# B&R Automation Studio project NAEUL004C00R13L518F00 (part 42)

#### Act_InitGlobal.st
```iecst
(** 2019-04-09 **)
ACTION Act_InitGlobal:

	(* Always Change If Project Change *)

	//Pass Data To Link
	p_bLinkOpsRun ACCESS p_OpsRun;

	p_bLinkDISafetyRlySig ACCESS p_DISafetyRlySig;
	p_bLinkDIConvClrSen ACCESS p_DIConvClrSen;
	p_bLinkDIPusherRetRS ACCESS p_DIPusherRetRS;
	p_bConvPusherReachedRetSlw ACCESS p_PshrConvPshrRetAllwTrav;
	p_eLinkLifterBtmStat ACCESS p_LifterBtmStat;
	p_eLinkLifterBtmStatus ACCESS p_LifterBtmStatus;
	p_eLinkLifter2Stat ACCESS p_Lifter2Stat;
	p_eLinkLifter2Status ACCESS p_Lifter2Status;

	//Pass Data To Internal Use
	p_udiRstErr ACCESS p_RstErrReset;
	p_bPrep ACCESS p_NtParamProjOutletShut2Prep;
	p_bUISimu ACCESS p_UISimuMod;
	p_bManual ACCESS p_UIMnlMod;
	p_bSimu ACCESS p_SimuRun;
	p_bTwoCtrlIn ACCESS p_NtParamOutShutterTwoCtrlIn;
	p_sProgNm ACCESS p_NtParamOutShutterProgNm;
	p_bExtSen ACCESS p_DIOutShutterCloseRS2;
	p_bRetSen ACCESS p_DIOutShutterOpenRS2;
	p_tExtTO ACCESS p_NtParamOutShutterExtTO;
	p_tRetTO ACCESS p_NtParamOutShutterRetTO;
	p_bNtSettingsLoadDone ACCESS p_StartupNtSettingsLoadDone;
	p_bNtParamProjLifter2Prep ACCESS p_NtParamProjLifter2Prep;
	(* Always Change If Project Change *)

END_ACTION
```

#### Act_LinkAction.st
```iecst
(** 2019-04-09 **)
ACTION Act_LinkAction:

	IF p_bLinkOpsRun = TRUE THEN
		IF p_bNtParamProjLifter2Prep = FALSE  THEN
			IF p_eLinkLifterBtmStat = LifterActIdle AND p_eLinkLifterBtmStatus <> Busy  THEN //
				p_eAct ACCESS p_OpsTravLifULOutletPneuAct2;
			ELSE
				p_eAct ACCESS ADR(eAct);
			END_IF
		ELSE
			IF p_eLinkLifterBtmStat = LifterActIdle AND p_eLinkLifterBtmStatus <> Busy AND p_eLinkLifter2Stat = LifterActIdle AND p_eLinkLifter2Status <> Busy  THEN // p_eLinkLifter2Status <> Busy
				p_eAct ACCESS p_OpsTravLifULOutletPneuAct2;
			ELSE
				p_eAct ACCESS ADR(eAct);
			END_IF
		END_IF
	ELSIF p_bManual = TRUE OR p_bUISimu THEN
		p_eAct ACCESS p_UIOutShutterAct2;
	ELSIF p_bSimu THEN
		p_eAct ACCESS p_Simu1OutShutterAct2;
	ELSE
		p_eAct ACCESS ADR(eAct);
	END_IF

END_ACTION
```

#### Act_LinkEn.st
```iecst
(** 2019-01-11 **)
ACTION Act_LinkEn:

	//Link bPrep, bEn & bDis
	p_bEn ACCESS p_NtParamCurtainSenPrep;

END_ACTION
```

#### Init.st
```iecst
(** 2019-03-25 **)
PROGRAM _INIT

	(* Always Change If Project Change *)

	//Pass Address To Global Address For External Use
	//Action, State & Status
	p_Pneu2SenOutShutterStat2		:= ADR(eStat);
	p_Pneu2SenOutShutterStatus2		:= ADR(eStatus);
	p_Pneu2SenOutShutterStatTxt2	:= ADR(sStatTxt);

	//Alarm
	p_Pneu2SenOutShutterAlmData2	:= ADR(tyAlmData);

	//Output
	p_Pneu2SenOutShutterExtCtrl2	:= ADR(bExtCtrl);
	p_Pneu2SenOutShutterRetCtrl2	:= ADR(bRetCtrl);
	p_Pneu2SenOutShutterTwoCtrlOut2	:= ADR(bTwoCtrlOut);
	p_Pneu2SenOutShutterExtended2	:= ADR(bExtended);
	p_Pneu2SenOutShutterRetracted2	:= ADR(bRetracted);

	(* Always Change If Project Change *)

END_PROGRAM
```

### Program Logical/Pneu/Pneu2SenOutShutter3

#### InputRef_Link.var
```iecst
(*2019-04-09*)
(**)
(*External*)
VAR
	p_bLinkOpsRun : REFERENCE TO BOOL;
END_VAR
(**)
VAR
	p_bLinkDISafetyRlySig : REFERENCE TO BOOL;
	p_bLinkDIConvClrSen : REFERENCE TO BOOL;
	p_bLinkDIPusherRetRS : REFERENCE TO BOOL;
	p_bConvPusherReachedRetSlw : REFERENCE TO BOOL;
	p_eLinkLifter2Stat : REFERENCE TO eLifterAction;
	p_eLinkLifter2Status : REFERENCE TO eFBStatus;
	p_eLinkLifterBtmStat : REFERENCE TO eLifterAction;
	p_eLinkLifterBtmStatus : REFERENCE TO eFBStatus;
END_VAR
```

#### Act_Alarm.st
```iecst
(** 2019-03-25 **)
ACTION Act_Alarm:

	//Error
	IF EDGEPOS(eStatus = Error) THEN

		tyAlmData.sProgNm		:= p_sProgNm;
		tyAlmData.udiCode		:= udiStatus;
		tyAlmData.eSeverity		:= AlmSeverityError;
		tyAlmData.udiRunTime	:= tyAlmData.udiRunTime + 1;
		tyAlmData.bAlm			:= TRUE;
		tyAlmData.udiModuleNum  := udiModuleNum;
		g_sPneu2SenProgNm		:= p_sProgNm;

		//Get Error Message
		IF tyAlmData.udiCode < 10000 OR tyAlmData.udiCode > 10099 THEN
			tyAlmData.sAlmMsg	:= 'Unknown';
			tyAlmData.sRcyMsg	:= 'Unknown';
		ELSE
			tyAlmData.sAlmMsg	:= a_tyAlmText[tyAlmData.udiCode].sAlmText;
			tyAlmData.sRcyMsg	:= a_tyAlmText[tyAlmData.udiCode].sRcyText;
		END_IF

		sStatTxt	:= tyAlmData.sAlmMsg;

	ELSIF bRstErr AND (tyAlmData.udiCode <> 0) THEN

		tyAlmData.udiCode	:= 0;
		tyAlmData.eSeverity	:= AlmSeverityNA;
		tyAlmData.sAlmMsg	:= '';
		tyAlmData.sRcyMsg	:= '';
		tyAlmData.bAlm			:= FALSE;
		sStatTxt	:= a_sStatText[eStat];

	END_IF

END_ACTION
```

#### Act_InitGlobal.st
```iecst
(** 2019-04-09 **)
ACTION Act_InitGlobal:

	(* Always Change If Project Change *)

	//Pass Data To Link
	p_bLinkOpsRun ACCESS p_OpsRun;

	p_bLinkDISafetyRlySig ACCESS p_DISafetyRlySig;
	p_bLinkDIConvClrSen ACCESS p_DIConvClrSen;
	p_bLinkDIPusherRetRS ACCESS p_DIPusherRetRS;
	p_bConvPusherReachedRetSlw ACCESS p_PshrConvPshrRetAllwTrav;
	p_eLinkLifterBtmStat ACCESS p_LifterBtmStat;
	p_eLinkLifterBtmStatus ACCESS p_LifterBtmStatus;
	p_eLinkLifter2Stat ACCESS p_Lifter2Stat;
	p_eLinkLifter2Status ACCESS p_Lifter2Status;

	//Pass Data To Internal Use
	p_udiRstErr ACCESS p_RstErrReset;
	p_bPrep ACCESS p_NtParamProjOutletShut3Prep;
	p_bUISimu ACCESS p_UISimuMod;
	p_bManual ACCESS p_UIMnlMod;
	p_bSimu ACCESS p_SimuRun;
	p_bTwoCtrlIn ACCESS p_NtParamOutShutterTwoCtrlIn;
	p_sProgNm ACCESS p_NtParamOutShutterProgNm;
	p_bExtSen ACCESS p_DIOutShutterCloseRS3;
	p_bRetSen ACCESS p_DIOutShutterOpenRS3;
	p_tExtTO ACCESS p_NtParamOutShutterExtTO;
	p_tRetTO ACCESS p_NtParamOutShutterRetTO;
	p_bNtSettingsLoadDone ACCESS p_StartupNtSettingsLoadDone;
	p_bNtParamProjLifter2Prep ACCESS p_NtParamProjLifter2Prep;
	(* Always Change If Project Change *)

END_ACTION
```

#### Act_Link.st
```iecst
(** 2019-03-29 **)
ACTION Act_Link:

	p_bExtSafetySen := (p_bLinkDIConvClrSen = FALSE) AND (p_bLinkDIPusherRetRS OR p_bConvPusherReachedRetSlw);

	IF p_bLinkDISafetyRlySig = FALSE THEN
		bExtCtrl	:= FALSE;
		bRetCtrl	:= FALSE;
		bExtended	:= FALSE;
		bRetracted	:= FALSE;
	END_IF

END_ACTION
```

#### Act_LinkAction.st
```iecst
(** 2019-04-09 **)
ACTION Act_LinkAction:

	IF p_bLinkOpsRun = TRUE THEN
		IF p_bNtParamProjLifter2Prep = FALSE  THEN
			IF p_eLinkLifterBtmStat = LifterActIdle AND p_eLinkLifterBtmStatus <> Busy  THEN //
				p_eAct ACCESS p_OpsTravLifULOutletPneuAct3;
			ELSE
				p_eAct ACCESS ADR(eAct);
			END_IF
		ELSE
			IF p_eLinkLifterBtmStat = LifterActIdle AND p_eLinkLifterBtmStatus <> Busy AND p_eLinkLifter2Stat = LifterActIdle AND p_eLinkLifter2Status <> Busy  THEN // p_eLinkLifter2Status <> Busy
				p_eAct ACCESS p_OpsTravLifULOutletPneuAct3;
			ELSE
				p_eAct ACCESS ADR(eAct);
			END_IF
		END_IF
	ELSIF p_bManual = TRUE OR p_bUISimu THEN
		p_eAct ACCESS p_UIOutShutterAct3;
	ELSIF p_bSimu THEN
		p_eAct ACCESS p_Simu1OutShutterAct3;
	ELSE
		p_eAct ACCESS ADR(eAct);
	END_IF

END_ACTION
```

### Program Logical/Pneu/Pneu2SenSelClamp1

#### Act_InitGlobal.st
```iecst
(** 2019-04-09 **)
ACTION Act_InitGlobal:

	(* Always Change If Project Change *)

	//Pass Data To Link
	p_bLinkOpsRun ACCESS p_OpsRun;

	p_bLinkDISafetyRlySig ACCESS p_DISafetyRlySig;

	//Pass Data To Internal Use
	p_udiRstErr ACCESS p_RstErrReset;
	p_bPrep ACCESS p_NtParamProjMagAutoVerifyPrep;
	p_bManual ACCESS p_UIMnlMod;
	p_bTwoCtrlIn ACCESS p_NtParamSelClamp1TwoCtrlIn;
	p_sProgNm ACCESS p_NtParamSelClamp1ProgNm;
	p_bExtSen ACCESS p_DIMag1SelUnclampRS;
//	p_bRetSen ACCESS p_DIOutShutterOpenRS;
	p_tExtTO ACCESS p_NtParamSelClamp1ExtDlyTm;
	p_tRetTO ACCESS p_NtParamSelClamp1RetDlyTm;
	p_bNtSettingsLoadDone ACCESS p_StartupNtSettingsLoadDone;

	(* Always Change If Project Change *)

END_ACTION
```

#### Act_LinkAction.st
```iecst
(** 2019-04-09 **)
ACTION Act_LinkAction:

	IF p_bLinkOpsRun = TRUE THEN
		p_eAct ACCESS p_OpsMagConvUL1StepSelClampCtrl;
	ELSIF p_bManual = TRUE THEN
		p_eAct ACCESS p_UIMagConvSelClp1Act;
	ELSE
		p_eAct ACCESS ADR(eAct);
	END_IF

END_ACTION
```

#### Init.st
```iecst
(** 2019-03-25 **)
PROGRAM _INIT

	(* Always Change If Project Change *)

	//Pass Address To Global Address For External Use
	//Action, State & Status
	p_PneuNoSenSelClamp1Stat		:= ADR(eStat);
	p_PneuNoSenSelClamp1Status		:= ADR(eStatus);
	p_PneuNoSenSelClamp1StatTxt		:= ADR(sStatTxt);

	//Alarm
	p_PneuNoSenSelClamp1AlmData		:= ADR(tyAlmData);

	//Output
	p_PneuNoSenSelClamp1ExtCtrl		:= ADR(bExtCtrl);
	p_PneuNoSenSelClamp1RetCtrl		:= ADR(bRetCtrl);
	p_PneuNoSenSelClamp1TwoCtrlOut	:= ADR(bTwoCtrlOut);
	p_PneuNoSenSelClamp1Extended	:= ADR(bExtended);
	p_PneuNoSenSelClamp1Retracted	:= ADR(bRetracted);

	(* Always Change If Project Change *)

END_PROGRAM
```

### Program Logical/Pneu/Pneu2SenSelClamp2

#### Act_Alarm.st
```iecst
(** 2019-03-25 **)
ACTION Act_Alarm:

	//Error
	IF EDGEPOS(eStatus = Error) THEN

		tyAlmData.sProgNm		:= p_sProgNm;
		tyAlmData.udiCode		:= udiStatus;
		tyAlmData.eSeverity		:= AlmSeverityError;
		tyAlmData.udiRunTime	:= tyAlmData.udiRunTime + 1;
		tyAlmData.bAlm			:= TRUE;
		tyAlmData.udiModuleNum  := udiModuleNum;
		g_sPneu2SenProgNm		:= p_sProgNm;

		//Get Error Message
		IF tyAlmData.udiCode < 10000 OR tyAlmData.udiCode > 10099 THEN
			tyAlmData.sAlmMsg	:= 'Unknown';
			tyAlmData.sRcyMsg	:= 'Unknown';
		ELSE
			tyAlmData.sAlmMsg	:= a_tyAlmText[tyAlmData.udiCode].sAlmText;
			tyAlmData.sRcyMsg	:= a_tyAlmText[tyAlmData.udiCode].sRcyText;
		END_IF

		sStatTxt	:= tyAlmData.sAlmMsg;

	ELSIF bRstErr AND (tyAlmData.udiCode <> 0) THEN

		tyAlmData.udiCode	:= 0;
		tyAlmData.eSeverity	:= AlmSeverityNA;
		tyAlmData.sAlmMsg	:= '';
		tyAlmData.sRcyMsg	:= '';
		tyAlmData.bAlm			:= FALSE;
		sStatTxt	:= a_sStatText[eStat];

	END_IF

END_ACTION
```

#### Act_InitGlobal.st
```iecst
(** 2029-04-09 **)
ACTION Act_InitGlobal:

	(* Always Change If Project Change *)

	//Pass Data To Link
	p_bLinkOpsRun ACCESS p_OpsRun;

	p_bLinkDISafetyRlySig ACCESS p_DISafetyRlySig;

	//Pass Data To Internal Use
	p_udiRstErr ACCESS p_RstErrReset;
	p_bPrep ACCESS p_NtParamProjMagAutoVerifyPrep;
	p_bManual ACCESS p_UIMnlMod;
	p_bTwoCtrlIn ACCESS p_NtParamSelClamp2TwoCtrlIn;
	p_sProgNm ACCESS p_NtParamSelClamp2ProgNm;
	p_bExtSen ACCESS p_DIMag2SelUnclampRS;
//	p_bRetSen ACCESS p_DIOutShutterOpenRS;
	p_tExtTO ACCESS p_NtParamSelClamp2ExtDlyTm;
	p_tRetTO ACCESS p_NtParamSelClamp2RetDlyTm;
	p_bNtSettingsLoadDone ACCESS p_StartupNtSettingsLoadDone;

	(* Always Change If Project Change *)

END_ACTION
```

#### Act_Link.st
```iecst
(** 2019-03-29 **)
ACTION Act_Link:

	IF p_bLinkDISafetyRlySig = FALSE THEN
		bExtCtrl	:= FALSE;
		bRetCtrl	:= FALSE;
		bExtended	:= FALSE;
		bRetracted	:= FALSE;
	END_IF

	p_bRetSen := NOT(p_bExtSen);
END_ACTION
```

#### Act_LinkAction.st
```iecst
(** 2019-04-09 **)
ACTION Act_LinkAction:

	IF p_bLinkOpsRun = TRUE THEN
		p_eAct ACCESS p_OpsMagConvUL2StepSelClampCtrl;
	ELSIF p_bManual = TRUE THEN
		p_eAct ACCESS p_UIMagConvSelClp2Act;
	ELSE
		p_eAct ACCESS ADR(eAct);
	END_IF

END_ACTION
```

#### Init.st
```iecst
(** 2029-03-25 **)
PROGRAM _INIT

	(* Always Change If Project Change *)

	//Pass Address To Global Address For External Use
	//Action, State & Status
	p_PneuNoSenSelClamp2Stat		:= ADR(eStat);
	p_PneuNoSenSelClamp2Status		:= ADR(eStatus);
	p_PneuNoSenSelClamp2StatTxt		:= ADR(sStatTxt);

	//Alarm
	p_PneuNoSenSelClamp2AlmData		:= ADR(tyAlmData);

	//Output
	p_PneuNoSenSelClamp2ExtCtrl		:= ADR(bExtCtrl);
	p_PneuNoSenSelClamp2RetCtrl		:= ADR(bRetCtrl);
	p_PneuNoSenSelClamp2TwoCtrlOut	:= ADR(bTwoCtrlOut);
	p_PneuNoSenSelClamp2Extended	:= ADR(bExtended);
	p_PneuNoSenSelClamp2Retracted	:= ADR(bRetracted);

	(* Always Change If Project Change *)

END_PROGRAM
```

### Program Logical/Pneu/Pneu2SenSelClamp3

#### Act_Alarm.st
```iecst
(** 2019-03-25 **)
ACTION Act_Alarm:

	//Error
	IF EDGEPOS(eStatus = Error) THEN

		tyAlmData.sProgNm		:= p_sProgNm;
		tyAlmData.udiCode		:= udiStatus;
		tyAlmData.eSeverity		:= AlmSeverityError;
		tyAlmData.udiRunTime	:= tyAlmData.udiRunTime + 1;
		tyAlmData.bAlm			:= TRUE;
		tyAlmData.udiModuleNum  := udiModuleNum;
		g_sPneu2SenProgNm		:= p_sProgNm;

		//Get Error Message
		IF tyAlmData.udiCode < 10000 OR tyAlmData.udiCode > 10099 THEN
			tyAlmData.sAlmMsg	:= 'Unknown';
			tyAlmData.sRcyMsg	:= 'Unknown';
		ELSE
			tyAlmData.sAlmMsg	:= a_tyAlmText[tyAlmData.udiCode].sAlmText;
			tyAlmData.sRcyMsg	:= a_tyAlmText[tyAlmData.udiCode].sRcyText;
		END_IF

		sStatTxt	:= tyAlmData.sAlmMsg;

	ELSIF bRstErr AND (tyAlmData.udiCode <> 0) THEN

		tyAlmData.udiCode	:= 0;
		tyAlmData.eSeverity	:= AlmSeverityNA;
		tyAlmData.sAlmMsg	:= '';
		tyAlmData.sRcyMsg	:= '';
		tyAlmData.bAlm			:= FALSE;
		sStatTxt	:= a_sStatText[eStat];

	END_IF

END_ACTION
```

#### Act_InitGlobal.st
```iecst
(** 2039-04-09 **)
ACTION Act_InitGlobal:

	(* Always Change If Project Change *)

	//Pass Data To Link
	p_bLinkOpsRun ACCESS p_OpsRun;

	p_bLinkDISafetyRlySig ACCESS p_DISafetyRlySig;

	//Pass Data To Internal Use
	p_udiRstErr ACCESS p_RstErrReset;
	p_bPrep ACCESS p_NtParamProjMagAutoVerifyPrep;
	p_bManual ACCESS p_UIMnlMod;
	p_bTwoCtrlIn ACCESS p_NtParamSelClamp3TwoCtrlIn;
	p_sProgNm ACCESS p_NtParamSelClamp3ProgNm;
	p_bExtSen ACCESS p_DIMag3SelUnclampRS;
//	p_bRetSen ACCESS p_DIOutShutterOpenRS;
	p_tExtTO ACCESS p_NtParamSelClamp3ExtDlyTm;
	p_tRetTO ACCESS p_NtParamSelClamp3RetDlyTm;
	p_bNtSettingsLoadDone ACCESS p_StartupNtSettingsLoadDone;

	(* Always Change If Project Change *)

END_ACTION
```

#### Act_LinkAction.st
```iecst
(** 2019-04-09 **)
ACTION Act_LinkAction:

	IF p_bLinkOpsRun = TRUE THEN
		p_eAct ACCESS p_OpsMagConvUL3StepSelClampCtrl;
	ELSIF p_bManual = TRUE THEN
		p_eAct ACCESS p_UIMagConvSelClp3Act;
	ELSE
		p_eAct ACCESS ADR(eAct);
	END_IF

END_ACTION
```

#### Init.st
```iecst
(** 2039-03-25 **)
PROGRAM _INIT

	(* Always Change If Project Change *)

	//Pass Address To Global Address For External Use
	//Action, State & Status
	p_PneuNoSenSelClamp3Stat		:= ADR(eStat);
	p_PneuNoSenSelClamp3Status		:= ADR(eStatus);
	p_PneuNoSenSelClamp3StatTxt		:= ADR(sStatTxt);

	//Alarm
	p_PneuNoSenSelClamp3AlmData		:= ADR(tyAlmData);

	//Output
	p_PneuNoSenSelClamp3ExtCtrl		:= ADR(bExtCtrl);
	p_PneuNoSenSelClamp3RetCtrl		:= ADR(bRetCtrl);
	p_PneuNoSenSelClamp3TwoCtrlOut	:= ADR(bTwoCtrlOut);
	p_PneuNoSenSelClamp3Extended	:= ADR(bExtended);
	p_PneuNoSenSelClamp3Retracted	:= ADR(bRetracted);

	(* Always Change If Project Change *)

END_PROGRAM
```

### Program Logical/Pneu/PneuNoSenInletStopper

#### Local.var
```iecst
(*2019-04-30*)
(**)
(*Local Action, State & Status*)
VAR
	eAct : ePneuAction := PneuActIdle;
	eStat : ePneuAction := PneuActIdle;
	eStatus : eFBStatus := Idle;
	udiStatus : UDINT := 0;
	sStatTxt : STRING[200] := '';
	a_sStatText : ARRAY[0..50] OF STRING[200] := ['Idling','Set All','Reset All','Set Extend','Set Retract','Extending','Retracting','Retracting From Extend Sensor To Middle Sensor','Retracting From Middle Sensor To Retract Sensor','Extending From Retract Sensor To Middle Sensor','Extending From Middle Sensor To Extend Sensor',40('')];
END_VAR
(**)
(*Local Alarm*)
VAR
	tyAlmData : tyAlmDat;
	a_tyAlmText : ARRAY[10000..10099] OF tyAlmTxt := [(sAlmText:='Safety Check Error While Extending',sRcyText:='Safety System Has Been Triggered. All Operations Are Disable. Remove the Obstacle That Triggered The Safety Interlock To Resume Operation.'),(sAlmText:='Extend Sensor On Checking Time Out While Extending',sRcyText:='Sensor Timeout Expired Before Operation Completed. Sensor Operation Is Abnormal. Solve The Error To Resume Operation. '),(sAlmText:='Retract Sensor Off Checking Time Out While Extending',sRcyText:='Sensor Timeout Expired Before Operation Completed. Sensor Operation Is Abnormal. Solve The Error To Resume Operation.'),(sAlmText:='Safety Check Error While Retracting',sRcyText:='Safety System Has Been Triggered. All Operations Are Disable. Remove the Obstacle That Triggered The Safety Interlock To Resume Operation.'),(sAlmText:='Retract Sensor On Checking Time Out While Retracting',sRcyText:='Sensor Timeout Expired Before Operation Completed. Sensor Operation Is Abnormal. Solve The Error To Resume Operation.'),(sAlmText:='Extend Sensor Off Checking Time Out While Retracting',sRcyText:='Sensor Timeout Expired Before Operation Completed. Sensor Operation Is Abnormal. Solve The Error To Resume Operation.'),94((0))];
END_VAR
(**)
(*Local Output*)
VAR
	bExtCtrl : BOOL;
	bRetCtrl : BOOL;
	bTwoCtrlOut : BOOL := FALSE;
	bExtended : BOOL := FALSE;
	bRetracted : BOOL := FALSE;
END_VAR
(**)
(*Local Input*)
VAR
	udiRstErr : UDINT := 0;
	bPrep : BOOL := TRUE;
	bEn : BOOL := TRUE;
	bDis : BOOL := FALSE;
	bManual : BOOL := FALSE;
	bTwoCtrlIn : BOOL := FALSE;
	bExtSafetySen : BOOL := TRUE;
	bRetSafetySen : BOOL := TRUE;
	sProgNm : STRING[15] := 'PneuNoSen';
	tExtDlyTm : TIME := T#1s;
	tRetDlyTm : TIME := T#1s;
	bNtSettingsLoadDone : BOOL := TRUE;
END_VAR
(**)
(*Local*)
VAR
	bRstErr : BOOL;
	udiRstErrOld : UDINT;
	bInitDone : BOOL;
	bInitialDone : BOOL;
	fbPneuExtChk : fbPneuNoSenExtChk;
	fbPneuRetChk : fbPneuNoSenRetChk;
	eStatOld : ePneuAction := PneuActIdle;
	bExtAllow : BOOL;
	bRetAllow : BOOL;
END_VAR
```

#### Act_Alarm.st
```iecst
(** 2019-03-25 **)
ACTION Act_Alarm:

	//Error
	IF EDGEPOS(eStatus = Error) THEN

		tyAlmData.sProgNm		:= p_sProgNm;
		tyAlmData.udiCode		:= udiStatus;
		tyAlmData.eSeverity		:= AlmSeverityError;
		tyAlmData.udiRunTime	:= tyAlmData.udiRunTime + 1;

		//Get Error Message
		IF tyAlmData.udiCode < 10000 OR tyAlmData.udiCode > 10099 THEN
			tyAlmData.sAlmMsg	:= 'Unknown';
			tyAlmData.sRcyMsg	:= 'Unknown';
		ELSE
			tyAlmData.sAlmMsg	:= a_tyAlmText[tyAlmData.udiCode].sAlmText;
			tyAlmData.sRcyMsg	:= a_tyAlmText[tyAlmData.udiCode].sRcyText;
		END_IF

		sStatTxt	:= tyAlmData.sAlmMsg;

	ELSIF bRstErr AND (tyAlmData.udiCode <> 0) THEN

		tyAlmData.udiCode	:= 0;
		tyAlmData.eSeverity	:= AlmSeverityNA;
		tyAlmData.sAlmMsg	:= '';
		tyAlmData.sRcyMsg	:= '';

		sStatTxt	:= a_sStatText[eStat];

	END_IF

END_ACTION
```

#### Act_InitGlobal.st
```iecst
(** 2019-04-09 **)
ACTION Act_InitGlobal:

	(* Always Change If Project Change *)

	//Pass Data To Link
	p_bLinkOpsRun ACCESS p_OpsRun;

	p_bLinkDISafetyRlySig ACCESS p_DISafetyRlySig;

	//Pass Data To Internal Use
	p_udiRstErr ACCESS p_RstErrReset;
	p_bPrep ACCESS p_NtParamProjInletStopperPrep;
	p_bDis ACCESS p_McParamInStopperDis;
	p_bManual ACCESS p_UIMnlMod;
	p_bTwoCtrlIn ACCESS p_NtParamInletStopperTwoCtrlIn;
	p_sProgNm ACCESS p_NtParamInletStopperProgNm;
	p_tExtDlyTm ACCESS p_NtParamInletStopperExtDlyTm;
	p_tRetDlyTm ACCESS p_NtParamInletStopperRetDlyTm;
	p_bNtSettingsLoadDone ACCESS p_StartupNtSettingsLoadDone;

	(* Always Change If Project Change *)

END_ACTION
```

#### Act_Link.st
```iecst
(** 2019-03-29 **)
ACTION Act_Link:

	IF p_bLinkDISafetyRlySig = FALSE THEN
		bExtCtrl	:= FALSE;
		bRetCtrl	:= FALSE;
		bExtended	:= FALSE;
		bRetracted	:= FALSE;
	END_IF

	//eAct
//	IF p_eConvDirection = ConvDirLToR THEN
//		bRetAllow			:= p_bLinkOpsLftConvStepUSCommTmr AND (p_bStopperUnBlkCtrl = FALSE);
//		bExtAllow			:= (p_bLinkOpsLftConvStepStandby AND (p_bLinkLftAWWidthPosDiff OR p_bLinkOpsLftAWStepMove)) OR (NOT p_bLinkLFFollowerUSAllow);
//		p_bEntBrdExtAllow	:= p_bLinkOpsInitLftConvStepInitCon OR p_bLinkOpsLftConvStepEntBrd OR (p_eLinkLftConvStat <> ConvActIdle);
//
//	END_IFs
//
//
//	IF p_bRetAllow AND (bRetCtrl = FALSE OR bExtCtrl = TRUE) THEN
//		eACT	:= StopperStepRet;
//	ELSIF p_bExtAllow AND (p_bStopperUnBlkCtrl = TRUE) THEN
//		eGotoStep	:= StopperStepExt;
//	ELSIF p_bEntBrdExtAllow AND (p_bStopperUnBlkCtrl = TRUE) THEN
//		eGotoStep	:= StopperStepEntBrdExt;
//		//					ELSE
//		//						bPaused	:= p_bStop OR p_bStep;
//	END_IF

END_ACTION
```

#### Act_LinkAction.st
```iecst
(** 2019-04-09 **)
ACTION Act_LinkAction:

	IF p_bLinkOpsRun = TRUE THEN
		p_eAct ACCESS p_OpsTravLifInletStprAct;
	ELSIF p_bManual = TRUE THEN
		p_eAct ACCESS p_UIInStopperAct;
	ELSE
		p_eAct ACCESS ADR(eAct);
	END_IF

END_ACTION
```

#### Act_LinkEn.st
```iecst
(** 2019-01-11 **)
ACTION Act_LinkEn:

	//Link bPrep, bEn & bDis
//	IF p_bDis = FALSE AND bExtCtrl = TRUE OR  bRetCtrl = FALSE
//		p_eAct := PneuActExt;
//	END_IF

END_ACTION
```

#### Cyclic.st
```iecst
(** 2019-03-29 **)
PROGRAM _CYCLIC

	IF bInitDone = FALSE THEN
		bInitDone	:= TRUE;

		Act_InitLocal;
		Act_InitGlobal;

	ELSIF bInitialDone = FALSE THEN
		IF p_bNtSettingsLoadDone = TRUE THEN
			bInitialDone	:= TRUE;

			Act_Initial;
		END_IF

	ELSE

		Act_RstErr;
		Act_LinkAction;
		Act_Action;
		Act_LinkEn;

		IF (p_bPrep = TRUE) AND (p_bEn = TRUE) AND (p_bDis = FALSE) THEN
			Act_Link;
			Act_Main;
		ELSE
			bExtCtrl	:= FALSE; //added
			bRetCtrl	:= TRUE; //added
			IF eStat <> PneuActIdle THEN
				IF eStat = PneuActSetExt OR eStat = PneuActExt THEN
					bExtended	:= TRUE;
					bRetracted	:= FALSE;
				ELSIF eStat = PneuActSetRet OR eStat = PneuActRet THEN
					bExtended	:= FALSE;
					bRetracted	:= TRUE;
				END_IF

				eStatus	:= Done;
			ELSE
				eStatus	:= Idle;
			END_IF
		END_IF

		Act_Alarm;

	END_IF

END_PROGRAM
```

#### Init.st
```iecst
(** 2019-03-25 **)
PROGRAM _INIT

	(* Always Change If Project Change *)

	//Pass Address To Global Address For External Use
	//Action, State & Status
	p_InletStopperStat				:= ADR(eStat);
	p_InletStopperStatus			:= ADR(eStatus);
	p_InletStopperStatTxt			:= ADR(sStatTxt);

	//Alarm
	p_InletStopperAlmData			:= ADR(tyAlmData);

	//Output
	p_InletStopperExtCtrl			:= ADR(bExtCtrl);
	p_InletStopperRetCtrl			:= ADR(bRetCtrl);
	p_InletStopperTwoCtrlOut		:= ADR(bTwoCtrlOut);
	p_InletStopperExtended			:= ADR(bExtended);
	p_InletStopperRetracted		:= ADR(bRetracted);

	(* Always Change If Project Change *)

END_PROGRAM
```

### Program Logical/Pneu/PneuNoSenStopperA

#### Act_InitGlobal.st
```iecst
(** 2019-04-09 **)
ACTION Act_InitGlobal:

	(* Always Change If Project Change *)

	//Pass Data To Link
	p_bLinkOpsRun ACCESS p_OpsRun;

	p_bLinkDISafetyRlySig ACCESS p_DISafetyRlySig;

	//Pass Data To Internal Use
	p_udiRstErr ACCESS p_RstErrReset;
	p_bPrep ACCESS p_NtParamProjStopperAPrep;
	p_bDis ACCESS p_McParamStopperADis;
	p_bManual ACCESS p_UIMnlMod;
	p_bTwoCtrlIn ACCESS p_NtParamStopperATwoCtrlIn;
	p_sProgNm ACCESS p_NtParamStopperAProgNm;
	p_tExtDlyTm ACCESS p_NtParamStopperAExtDlyTm;
	p_tRetDlyTm ACCESS p_NtParamStopperARetDlyTm;
	p_bNtSettingsLoadDone ACCESS p_StartupNtSettingsLoadDone;

	(* Always Change If Project Change *)

END_ACTION
```

#### Act_LinkAction.st
```iecst
(** 2019-04-09 **)
ACTION Act_LinkAction:

	IF p_bLinkOpsRun = TRUE THEN
		p_eAct ACCESS p_OpsTravLifULStopperAct1;
	ELSIF p_bManual = TRUE THEN
		p_eAct ACCESS p_UIStopperAAct;
	ELSE
		p_eAct ACCESS ADR(eAct);
	END_IF

END_ACTION
```

#### Init.st
```iecst
(** 2019-03-25 **)
PROGRAM _INIT

	(* Always Change If Project Change *)

	//Pass Address To Global Address For External Use
	//Action, State & Status
	p_PneuNoSenStopperAStat			:= ADR(eStat);
	p_PneuNoSenStopperAStatus		:= ADR(eStatus);
	p_PneuNoSenStopperAStatTxt		:= ADR(sStatTxt);

	//Alarm
	p_PneuNoSenStopperAAlmData		:= ADR(tyAlmData);

	//Output
	p_PneuNoSenStopperAExtCtrl		:= ADR(bExtCtrl);
	p_PneuNoSenStopperARetCtrl		:= ADR(bRetCtrl);
	p_PneuNoSenStopperATwoCtrlOut	:= ADR(bTwoCtrlOut);
	p_PneuNoSenStopperAExtended		:= ADR(bExtended);
	p_PneuNoSenStopperARetracted	:= ADR(bRetracted);

	(* Always Change If Project Change *)

END_PROGRAM
```

### Program Logical/Pneu/PneuNoSenStopperB (IEC, version 1.00.0)

#### Init.st - Change By Project
```iecst
(** 2019-03-25 **)
PROGRAM _INIT

	(* Always Change If Project Change *)

	//Pass Address To Global Address For External Use
	//Action, State & Status
	p_PneuNoSenStopperBStat			:= ADR(eStat);
	p_PneuNoSenStopperBStatus		:= ADR(eStatus);
	p_PneuNoSenStopperBStatTxt		:= ADR(sStatTxt);

	//Alarm
	p_PneuNoSenStopperBAlmData		:= ADR(tyAlmData);

	//Output
	p_PneuNoSenStopperBExtCtrl		:= ADR(bExtCtrl);
	p_PneuNoSenStopperBRetCtrl		:= ADR(bRetCtrl);
	p_PneuNoSenStopperBTwoCtrlOut	:= ADR(bTwoCtrlOut);
	p_PneuNoSenStopperBExtended		:= ADR(bExtended);
	p_PneuNoSenStopperBRetracted	:= ADR(bRetracted);

	(* Always Change If Project Change *)

END_PROGRAM
```

#### Act_InitGlobal.st - Change By Project
```iecst
(** 2019-04-09 **)
ACTION Act_InitGlobal:

	(* Always Change If Project Change *)

	//Pass Data To Link
	p_bLinkOpsRun ACCESS p_OpsRun;

	p_bLinkDISafetyRlySig ACCESS p_DISafetyRlySig;

	//Pass Data To Internal Use
	p_udiRstErr ACCESS p_RstErrReset;
	p_bPrep ACCESS p_NtParamProjStopperBPrep;
	p_bDis ACCESS p_McParamStopperBDis;
	p_bManual ACCESS p_UIMnlMod;
	p_bTwoCtrlIn ACCESS p_NtParamStopperBTwoCtrlIn;
	p_sProgNm ACCESS p_NtParamStopperBProgNm;
	p_tExtDlyTm ACCESS p_NtParamStopperBExtDlyTm;
	p_tRetDlyTm ACCESS p_NtParamStopperBRetDlyTm;
	p_bNtSettingsLoadDone ACCESS p_StartupNtSettingsLoadDone;

	(* Always Change If Project Change *)

END_ACTION
```

#### Act_LinkAction.st - Change By Project
```iecst
(** 2019-04-09 **)
ACTION Act_LinkAction:

	IF p_bLinkOpsRun = TRUE THEN
		p_eAct ACCESS p_OpsTravLifULStopperAct2;
	ELSIF p_bManual = TRUE THEN
		p_eAct ACCESS p_UIStopperBAct;
	ELSE
		p_eAct ACCESS ADR(eAct);
	END_IF

END_ACTION
```

#### Act_Alarm.st - Do Not Change!!!
```iecst
(** 2019-03-25 **)
ACTION Act_Alarm:

	//Error
	IF EDGEPOS(eStatus = Error) THEN

		tyAlmData.sProgNm		:= p_sProgNm;
		tyAlmData.udiCode		:= udiStatus;
		tyAlmData.eSeverity		:= AlmSeverityError;
		tyAlmData.udiRunTime	:= tyAlmData.udiRunTime + 1;
		tyAlmData.bAlm			:= TRUE;
		tyAlmData.udiModuleNum  := udiModuleNum;
		g_sPneuNoSenProgNm		:= p_sProgNm;;

		//Get Error Message
		IF tyAlmData.udiCode < 10000 OR tyAlmData.udiCode > 10099 THEN
			tyAlmData.sAlmMsg	:= 'Unknown';
			tyAlmData.sRcyMsg	:= 'Unknown';
		ELSE
			tyAlmData.sAlmMsg	:= a_tyAlmText[tyAlmData.udiCode].sAlmText;
			tyAlmData.sRcyMsg	:= a_tyAlmText[tyAlmData.udiCode].sRcyText;
		END_IF

		sStatTxt	:= tyAlmData.sAlmMsg;

	ELSIF bRstErr AND (tyAlmData.udiCode <> 0) THEN

		tyAlmData.udiCode	:= 0;
		tyAlmData.eSeverity	:= AlmSeverityNA;
		tyAlmData.sAlmMsg	:= '';
		tyAlmData.sRcyMsg	:= '';
		tyAlmData.bAlm			:= FALSE;
		sStatTxt	:= a_sStatText[eStat];

	END_IF

END_ACTION
```

### Program Logical/Pneu/PneuNoSenStopperC

#### Act_InitGlobal.st
```iecst
(** 2019-04-09 **)
ACTION Act_InitGlobal:

	(* Always Change If Project Change *)

	//Pass Data To Link
	p_bLinkOpsRun ACCESS p_OpsRun;

	p_bLinkDISafetyRlySig ACCESS p_DISafetyRlySig;

	//Pass Data To Internal Use
	p_udiRstErr ACCESS p_RstErrReset;
	p_bNtSettingsLoadDone ACCESS p_StartupNtSettingsLoadDone;

	(* Always Change If Project Change *)

END_ACTION
```

#### Act_LinkAction.st
```iecst
(** 2019-04-09 **)
ACTION Act_LinkAction:

	IF p_bLinkOpsRun = TRUE THEN
		p_eAct ACCESS p_OpsTravLifULStopperAct3;
	ELSE
		p_eAct ACCESS ADR(eAct);
	END_IF

END_ACTION
```

#### Init.st
```iecst
(** 2019-03-25 **)
PROGRAM _INIT

	(* Always Change If Project Change *)

	//Physical Configuration
	bPrep	:= FALSE;

	//Pass Address To Global Address For External Use
	//Action, State & Status
	p_PneuNoSenStopperCStat			:= ADR(eStat);
	p_PneuNoSenStopperCStatus		:= ADR(eStatus);
	p_PneuNoSenStopperCStatTxt		:= ADR(sStatTxt);

	//Alarm
	p_PneuNoSenStopperCAlmData		:= ADR(tyAlmData);

	//Output
	p_PneuNoSenStopperCExtCtrl		:= ADR(bExtCtrl);
	p_PneuNoSenStopperCRetCtrl		:= ADR(bRetCtrl);
	p_PneuNoSenStopperCTwoCtrlOut	:= ADR(bTwoCtrlOut);
	p_PneuNoSenStopperCExtended		:= ADR(bExtended);
	p_PneuNoSenStopperCRetracted	:= ADR(bRetracted);

	(* Always Change If Project Change *)

END_PROGRAM
```

### MagConv2Clp.typ - Change By Project
```iecst
(*2019-10-30*)
(**)
(*Action*)

TYPE
	eMagConv2ClpAction :
		(
		MagConv2ClpActIdle,
		MagConv2ClpActInit,
		MagConv2ClpActInitStopClp,
		MagConv2ClpActInitClpStop,
		MagConv2ClpActEnt,
		MagConv2ClpActEntStopClp,
		MagConv2ClpActEntClpStop,
		MagConv2ClpActPreExit,
		MagConv2ClpActPreExitClpr,
		MagConv2ClpActPreExitClpr1,
		MagConv2ClpActExit,
		MagConv2ClpActExit1,
		MagConv2ClpActExitClpr,
		MagConv2ClpActExit1Clpr,
		MagConv2ClpActFixClprSetAll,
		MagConv2ClpActFixClprRstAll,
		MagConv2ClpActFixClprSetClamp,
		MagConv2ClpActFixClprSetUnclamp,
		MagConv2ClpActFixClprClamp,
		MagConv2ClpActFixClprUnclamp,
		MagConv2ClpActRmtClprSetAll,
		MagConv2ClpActRmtClprRstAll,
		MagConv2ClpActRmtClprSetClamp,
		MagConv2ClpActRmtClprSetUnclamp,
		MagConv2ClpActRmtClprClamp,
		MagConv2ClpActRmtClprUnclamp,
		MagConv2ClpActStop,
		MagConv2ClpActStopClpr,
		MagConv2ClpActSetMtrSigOnOrLToR,
		MagConv2ClpActSetMtrDirOrRToL,
		MagConv2ClpActRstMtrSigOnOrLToR,
		MagConv2ClpActRstMtrDirOrRToL,
		MagConv2ClpActSetMtrAll,
		MagConv2ClpActRstMtrAll
		);
END_TYPE

(**)

TYPE
	tyMagConv2Clp : 	STRUCT
		In : tyMagConv2ClpIn1;
		Out : tyMagConv2ClpOut1;
	END_STRUCT;
	tyMagConv2ClpIn1 : 	STRUCT
		bLinkDISafetyRlySig : BOOL;
		bLinkMagSmallSen : BOOL;
		bLinkMagLargeSen : BOOL;
		bLinkFixClprUnClampSen : BOOL;
		bLinkFixClprClampSen : BOOL;
		bLinkRmtClprUnclampSen : BOOL;
		bLinkFixClprMagDetectSen : BOOL;
		bLinkFixClprMagDetectSenPrep : BOOL;
		bLinkMagOpsStepMagFullExit : BOOL;
		bLinkDIMagEntSen : BOOL;
		bWidthChkSen : BOOL;
		bWidthChkInterrupt : BOOL;
		bLinkNtParamMagModelAutoVerify : BOOL;
		udiRstErr : UDINT;
		bPrep : BOOL;
		bEn : BOOL;
		bDis : BOOL;
		bManual : BOOL;
		bOnDirMod : BOOL;
		diInitTm : DINT;
		tMtrOffDlyTm : TIME;
		diTxInTimeOut : DINT;
		diTxOutTimeOut : DINT;
		eDirection : eConvDir;
		sProgNm : STRING[15];
		tClprClampTO : TIME;
		tClprUnclampTO : TIME;
		bLeftSen : BOOL;
		bRightSen : BOOL;
		bFixClprUnclampSen : BOOL;
		bRmtClprUnclampSen : BOOL;
		bFixClprClampSen : BOOL;
		bRmtClprClampSen : BOOL;
		bFixClprClampSafetySen : BOOL;
		bFixClprUnclampSafetySen : BOOL;
		bRmtClprClampSafetySen : BOOL;
		bRmtClprUnclampSafetySen : BOOL;
		bWidthChkPrep : BOOL;
	END_STRUCT;
	tyMagConv2ClpOut1 : 	STRUCT
		eStat : eMagConv2ClpAction;
		eStatus : eFBStatus;
		sStatTxt : STRING[200];
		tyAlmData : tyAlmDat;
		bHvMag : BOOL;
		bMtrSigOnOrLToR : BOOL;
		bMtrDirOrRToL : BOOL;
		bFixClprClampCtrl : BOOL;
		bRmtClprClampCtrl : BOOL;
		bClprTwoOutputControl : BOOL;
		bRmtClprUnClampCtrl : BOOL;
		bFixClprUnClampCtrl : BOOL;
	END_STRUCT;
END_TYPE
```

### MagConv2Clp.var - Change By Project
```iecst
VAR
	g_tyMagConv2Clp1 : tyMagConv2ClpOut1; (*OutletShutter*)
	g_tyMagConv2Clp2 : tyMagConv2ClpOut1; (*OutletShutter*)
	g_tyMagConv2Clp3 : tyMagConv2ClpOut1; (*OutletShutter*)
END_VAR
```

### Program Logical/MagConv_LiftnTrav/MagConv2Clp1 (IEC, version 1.00.0) - 1.00.0 - NtConv v5.00.0 , NtPneu v5.00.0

#### Init.st - Change By Project
```iecst
(** 2019-10-30 **)
PROGRAM _INIT

	(* Always Change If Project Change *)

	//Pass Address To Global Address For External Use
	//Action, State & Status
	p_MagConv2Clp1Stat				:= ADR(eStat);
	p_MagConv2Clp1Status			:= ADR(eStatus);
	p_MagConv2Clp1StatTxt			:= ADR(sStatTxt);

	//Alarm
	p_MagConv2Clp1AlmData			:= ADR(tyAlmData);

	//Output
	p_MagConv2Clp1HvMag				:= ADR(bHvMag);
	p_MagConv2Clp1MtrSigOnOrLToR	:= ADR(bMtrSigOnOrLToR);
	p_MagConv2Clp1MtrDirOrRToL		:= ADR(bMtrDirOrRToL);

	p_MagConv2Clp1FixClprClampCtrl	:= ADR(bFixClprClampCtrl);
	p_MagConv2Clp1RmtClprClampCtrl	:= ADR(bRmtClprClampCtrl);
	p_MagConv2Clp1ClprTwoOutputCtrl	:= ADR(bClprTwoOutputControl);

	(* Always Change If Project Change *)

END_PROGRAM
```

#### Act_InitGlobal.st - Change By Project
```iecst
(** 2019-10-30 **)
ACTION Act_InitGlobal:

	(* Always Change If Project Change *)

	//Pass Data To Link
	p_bLinkOpsRun ACCESS p_OpsRun;

	p_bLinkDISafetyRlySig ACCESS p_DISafetyRlySig;

	p_bLinkMagSmallSen ACCESS p_DIMagConvSmallMagSen1;
	p_bLinkMagLargeSen ACCESS p_DIMagConvLargeMagSen1;
	p_bLinkFixClprUnClampSen ACCESS p_DIMag1FixedUnclampRS;
	p_bLinkFixClprClampSen ACCESS p_DIMag1FixedClampRS; // Pneumatic Clamp Reed Switch
	p_bLinkFixClprMagDetectSen ACCESS p_DIMag1FixedClampSen; // Clamping Done Before Pneumatic Clamp Reed Switch for special Condition
	p_bLinkFixClprMagDetectSenPrep ACCESS p_NtParamProjFixClpMagDSenPrep; // Fixed Clamp Detect Sensor Prep before Clamp RS

	p_bLinkMagOpsStepMagFullExit ACCESS p_OpsMagConvUL1MagFullExit;
	p_bLinkDIMagEntSen ACCESS p_DIMagConvEntSen1;
	p_bLinkDO ACCESS p_DO;

	p_bWidthChkSen ACCESS p_NtParamCurtainSenPrep;
	p_bWidthChkInterrupt ACCESS p_DICurtainSen;

	p_bLinkNtParamMagModelAutoVerify ACCESS p_NtParamProjMagAutoVerifyPrep;
	p_tyDISettings ACCESS p_NtParamDISettings;
	p_bLinkFixClprClampSen ACCESS ADR(bFixClprClampSen);//p_DIMag1FixedSideDetect;//p_DIMag1FixedClampRS; //initLocal at 1st

	//Pass Data To Internal Use
	p_udiRstErr ACCESS p_RstErrReset;
	p_bPrep ACCESS p_NtParamProjMag1ConvPrep;
	p_bManual ACCESS p_UIMnlMod;
	p_bOnDirMod ACCESS p_NtParamMagConv1OnDirMod;
	p_diInitTm ACCESS p_McParamMag1ConvRunTmOut;
	p_tMtrOffDlyTm ACCESS p_NtParamMagConv1MtrOffDlyTm;
	p_diTxInTimeOut ACCESS p_McParamMag1ConvRunTmOut;
	p_diTxOutTimeOut ACCESS p_McParamMag1ConvRunTmOut;
	p_eDirection ACCESS p_NtParamProjMagConvDir;
	p_sProgNm ACCESS p_NtParamMagConv1ProgNm;
	p_tClprClampTO ACCESS p_NtParamMagConv1ClprClampTO;
	p_tClprUnclampTO ACCESS p_NtParamMagConv1ClprUnclampTO;
//	p_bLeftSen ACCESS p_DIMagPresentSen1;
	p_bRightSen	ACCESS p_DIMagPresentSen1;

	p_bNtSettingsLoadDone ACCESS p_StartupNtSettingsLoadDone;

	(* Always Change If Project Change *)

END_ACTION
```

#### InputRef_Link.var - Change By Project
```iecst
(*2019-10-30*)
(**)
VAR
	p_bLinkOpsRun : REFERENCE TO BOOL;
END_VAR
(**)
VAR
	p_bLinkDISafetyRlySig : REFERENCE TO BOOL;
	p_bLinkMagSmallSen : REFERENCE TO BOOL;
	p_bLinkMagLargeSen : REFERENCE TO BOOL;
	p_bLinkFixClprUnClampSen : REFERENCE TO BOOL;
	p_bLinkFixClprClampSen : REFERENCE TO BOOL;
	p_bLinkFixClprMagDetectSen : REFERENCE TO BOOL;
	p_bLinkFixClprMagDetectSenPrep : REFERENCE TO BOOL;
	p_bLinkMagOpsStepMagFullExit : REFERENCE TO BOOL;
	p_bLinkDIMagEntSen : REFERENCE TO BOOL;
	p_bLinkDIMagPresentSen : REFERENCE TO BOOL;
	p_bLinkDO : REFERENCE TO tyDigitalOutput;
	p_bLinkNtParamMagModelAutoVerify : REFERENCE TO BOOL;
	p_tyDISettings : REFERENCE TO tyDigitalInputSettings;
END_VAR
```

#### Act_LinkAction.st - Change By Project
```iecst
(** 2019-10-30 **)
ACTION Act_LinkAction:

	IF p_bLinkOpsRun = TRUE THEN
		p_eAct ACCESS p_OpsMagConvUL1MagConv2ClpAct;
	ELSIF p_bManual = TRUE THEN
		p_eAct ACCESS p_UIMagConv2Clp1Act;
	ELSE
		p_eAct ACCESS ADR(eAct);
	END_IF

END_ACTION
```

#### Act_Link.st - Change By Project
```iecst
(** 2019-10-30 **)
ACTION Act_Link:

	IF tylocalMagConv2Clp.In.bLinkDISafetyRlySig = FALSE THEN
		tylocalMagConv2Clp.Out.bFixClprClampCtrl	:= FALSE;
		tylocalMagConv2Clp.Out.bRmtClprClampCtrl	:= FALSE;
		tylocalMagConv2Clp.Out.bFixClprUnClampCtrl	:= FALSE;
		tylocalMagConv2Clp.Out.bRmtClprUnClampCtrl	:= FALSE;
	END_IF

	tylocalMagConv2Clp.In.bFixClprUnclampSen :=  tylocalMagConv2Clp.In.bLinkFixClprUnClampSen;
	tylocalMagConv2Clp.In.bRmtClprUnclampSen := tylocalMagConv2Clp.In.bLinkRmtClprUnclampSen;

	IF tylocalMagConv2Clp.In.bLinkNtParamMagModelAutoVerify THEN
		fbSmallLargeSenDlyTm(IN:= tylocalMagConv2Clp.In.bLinkMagSmallSen OR tylocalMagConv2Clp.In.bLinkMagLargeSen);
		IF fbSmallLargeSenDlyTm.Q THEN
			tylocalMagConv2Clp.In.bFixClprClampSen := TRUE;
		ELSE
			tylocalMagConv2Clp.In.bFixClprClampSen := FALSE;
		END_IF
	ELSIF tylocalMagConv2Clp.In.tyDISettings.diMag1FixedClampSen = 0 THEN
		tylocalMagConv2Clp.In.bFixClprClampSen := tylocalMagConv2Clp.In.bLinkFixClprClampSen; //Normal Pneumatic Clamping RS.
	ELSE
		IF tylocalMagConv2Clp.Out.eStat = MagConv2ClpActInitStopClp AND usiStep = 3 OR
			tylocalMagConv2Clp.Out.eStat = MagConv2ClpActEntStopClp AND usiStep = 2 OR
			tylocalMagConv2Clp.Out.eStat = MagConv2ClpActFixClprClamp OR tylocalMagConv2Clp.Out.eStat = MagConv2ClpActFixClprUnclamp THEN //during fix clamp
			fbFixClpExtChkTm(IN:=TRUE);
			IF fbFixClpExtChkTm.Q THEN
				fbFixClpExtChkTm(IN:=FALSE);
				tylocalMagConv2Clp.In.bFixClprClampSen := tylocalMagConv2Clp.In.bLinkFixClprMagDetectSen;
			END_IF
		ELSIF	tylocalMagConv2Clp.Out.eStat = MagConv2ClpActInitStopClp AND usiStep = 4 OR
			tylocalMagConv2Clp.Out.eStat = MagConv2ClpActEntStopClp AND usiStep = 3 OR
			tylocalMagConv2Clp.Out.eStat = MagConv2ClpActRmtClprClamp OR tylocalMagConv2Clp.Out.eStat = MagConv2ClpActRmtClprUnclamp THEN //during remote clamp
			fbRmtClpExtChkTm(IN:=TRUE);
			IF fbRmtClpExtChkTm.Q THEN
				fbRmtClpExtChkTm(IN:=FALSE);
				tylocalMagConv2Clp.In.bRmtClprClampSen := tylocalMagConv2Clp.Out.bRmtClprClampCtrl;
			END_IF
		ELSE
			fbFixClpExtChkTm(IN:=FALSE);
			fbRmtClpExtChkTm(IN:=FALSE);
			tylocalMagConv2Clp.In.bFixClprClampSen := FALSE;
			tylocalMagConv2Clp.In.bRmtClprClampSen := FALSE;
		END_IF
	END_IF

	IF tylocalMagConv2Clp.In.bLinkMagOpsStepMagFullExit THEN
		fbLeftSenDelayTm(IN:= TRUE, PT:=  T#3000ms);
		IF fbLeftSenDelayTm.Q THEN
			tylocalMagConv2Clp.In.bLeftSen := tylocalMagConv2Clp.In.bLinkDIMagEntSen;
		END_IF
	ELSE
		tylocalMagConv2Clp.In.bLeftSen := tylocalMagConv2Clp.In.bLinkDIMagEntSen;
		fbLeftSenDelayTm(IN:= FALSE);
	END_IF

END_ACTION
```

#### Act_Initial.st - Do Not Change!!!
```iecst
(** 2019-10-30 **)
ACTION Act_Initial:

	//Initial
	sStatTxt	:= a_sStatText[eStat];

	fbInit.bOnDirMod	:= p_bOnDirMod;
	fbInit.bStartSen	:= TRUE;
	fbInit.tMtrOffDlyTm	:= p_tMtrOffDlyTm;
	fbInit(bEn := FALSE);

	fbEnt.bOnDirMod		:= p_bOnDirMod;
	fbEnt.bStartSen		:= TRUE;
	fbEnt.tMtrOffDlyTm	:= p_tMtrOffDlyTm;
	fbEnt(bEn := FALSE);

	fbPreExit.bOnDirMod		:= p_bOnDirMod;
	fbPreExit.bStartSen		:= TRUE;
	fbPreExit.tMtrOffDlyTm	:= p_tMtrOffDlyTm;
	fbPreExit(bEn := FALSE);

	fbExit.bOnDirMod	:= p_bOnDirMod;
	fbExit.bStartSen	:= TRUE;
	fbExit.tMtrOffDlyTm	:= p_tMtrOffDlyTm;
	fbExit(bEn := FALSE);

	fbExit1.bOnDirMod		:= p_bOnDirMod;
	fbExit1.bStartSen		:= TRUE;
	fbExit1.tMtrOffDlyTm	:= p_tMtrOffDlyTm;
	fbExit1(bEn := FALSE);

	fbStop(bEn := FALSE);

	fbFixClprClampChk.tTimeOut	:= p_tClprClampTO;
	fbFixClprClampChk(bEn := FALSE);

	fbFixClprUnclampChk.tTimeOut	:= p_tClprUnclampTO;
	fbFixClprUnclampChk(bEn := FALSE);

	fbRmtClprClampChk.tTimeOut	:= p_tClprClampTO;
	fbRmtClprClampChk(bEn := FALSE);

	fbRmtClprUnclampChk.tTimeOut	:= p_tClprUnclampTO;
	fbRmtClprUnclampChk(bEn := FALSE);

	fbClprDlyTm.PT	:= p_tMtrOffDlyTm / 2;
	fbClprDlyTm(IN := FALSE);

END_ACTION
```

#### Act_Action.st - Do Not Change!!!
```iecst
(** 2019-10-30 **)
ACTION Act_Action:

	//Reset Error
	IF (eStatus = Error) AND bRstErr THEN
		p_eAct	:= MagConv2ClpActIdle;
		eStat	:= MagConv2ClpActIdle;
	END_IF

	//Set p_eAct
	IF eStatus = Idle OR eStatus = Busy OR eStatus = Done THEN
		eStat	:= p_eAct;
	END_IF

END_ACTION
```

#### Act_Main.st - Do Not Change!!!
```iecst
(** 2019-10-30 **)
ACTION Act_Main:

	IF eStatOld <> eStat THEN
		fbInit(bEn := FALSE);
		fbEnt(bEn := FALSE);
		fbPreExit(bEn := FALSE);
		fbExit(bEn := FALSE);
		fbExit1(bEn := FALSE);
		fbStop(bEn := FALSE);
		fbFixClprClampChk(bEn := FALSE);
		fbFixClprUnclampChk(bEn := FALSE);
		fbRmtClprClampChk(bEn := FALSE);
		fbRmtClprUnclampChk(bEn := FALSE);
		fbClprDlyTm(IN := FALSE);
		fbFixClprDly(IN := FALSE);
		fbWidthChk(IN := FALSE);

		IF eStatOld <> MagConv2ClpActIdle
			AND eStatOld <> MagConv2ClpActSetMtrSigOnOrLToR
			AND eStatOld <> MagConv2ClpActSetMtrDirOrRToL
			AND eStatOld <> MagConv2ClpActRstMtrSigOnOrLToR
			AND eStatOld <> MagConv2ClpActRstMtrDirOrRToL
			AND eStatOld <> MagConv2ClpActSetMtrAll
			AND eStatOld <> MagConv2ClpActRstMtrAll THEN

			bMtrSigOnOrLToR	:= FALSE;
			bMtrDirOrRToL	:= FALSE;

		END_IF

		usiStep		:= 0;
		usiSubStep	:= 0;
		bReachEnd	:= FALSE;

		sStatTxt	:= a_sStatText[eStat];

		eStatOld	:= eStat;

		eStatus		:= Busy;
	END_IF

	//Main
	CASE eStat OF

		MagConv2ClpActIdle:
			IF EDGENEG(p_bManual) THEN
				bMtrSigOnOrLToR	:= FALSE;
				bMtrDirOrRToL	:= FALSE;
			END_IF

			eStatus	:= Idle;

		MagConv2ClpActInit:
			IF eStatus = Idle OR eStatus = Busy THEN

				eStatus	:= Busy;

				//Magazine Conveyor Init Run
				//Detect Have Magazine
				IF p_bLeftSen OR p_bRightSen THEN
					bHvMag	:= TRUE;
				ELSE
					bHvMag	:= FALSE;
				END_IF

				fbInit.bConvLToR	:= (p_eDirection = ConvDirLToR) OR (p_eDirection = ConvDirLToL);
				fbInit.tTxDlyTm		:= DINT_TO_TIME(p_diInitTm);

				IF fbInit.bConvLToR = TRUE THEN
					fbInit.bEndSen	:= p_bRightSen;
				ELSE
					fbInit.bEndSen	:= p_bLeftSen;
				END_IF

				fbInit(bEn := TRUE);

				bMtrSigOnOrLToR	:= fbInit.bMtrSigOnOrLToR;
				bMtrDirOrRToL	:= fbInit.bMtrDirOrRToL;

				IF fbInit.udiStatus = 0 THEN
					IF fbInit.bConvLToR = TRUE THEN
						IF bHvMag = TRUE AND p_bRightSen = FALSE THEN
							udiStatus	:= 10000;	//Magazine Detected But Not Present At Outlet Sensor (L - R) While Magazine Conveyor Initial
							eStatus		:= Error;
						ELSE
							eStatus	:= Done;
						END_IF
					ELSE
						IF bHvMag = TRUE AND p_bLeftSen = FALSE THEN
							udiStatus	:= 10001;	//Magazine Detected But Not Present At Outlet Sensor (R - L) While Magazine Conveyor Initial
							eStatus		:= Error;
						ELSE
							eStatus	:= Done;
						END_IF
					END_IF
				ELSIF fbInit.udiStatus < 65534 THEN
					udiStatus	:= fbInit.udiStatus;
					eStatus		:= Error;
				END_IF
			END_IF

		MagConv2ClpActInitStopClp:
			IF eStatus = Idle OR eStatus = Busy THEN

				eStatus	:= Busy;

				CASE usiStep OF
					0:	//Unclamp
						bFixClprClampCtrl	:= FALSE;
						bRmtClprClampCtrl	:= FALSE;

						fbFixClprUnclampChk.bExtSen		:= p_bFixClprClampSen;
						fbFixClprUnclampChk.bRetSen		:= p_bFixClprUnclampSen;
						fbFixClprUnclampChk.bRetSafety	:= p_bFixClprUnclampSafetySen;
						fbFixClprUnclampChk(bEn := TRUE);

						fbRmtClprUnclampChk.bExtSen		:= p_bRmtClprClampSen;
						fbRmtClprUnclampChk.bRetSen		:= p_bRmtClprUnclampSen;
						fbRmtClprUnclampChk.bRetSafety	:= p_bRmtClprUnclampSafetySen;
						fbRmtClprUnclampChk(bEn := TRUE);

						IF fbFixClprUnclampChk.udiStatus = 0 AND fbRmtClprUnclampChk.udiStatus = 0 THEN
							usiStep	:= 1;
						ELSIF (fbFixClprUnclampChk.udiStatus > 0 AND fbFixClprUnclampChk.udiStatus < 65534) OR (fbRmtClprUnclampChk.udiStatus > 0 AND fbRmtClprUnclampChk.udiStatus < 65534) THEN
							bFixClprClampCtrl	:= TRUE;
							bRmtClprClampCtrl	:= TRUE;

							eStatus	:= Error;

							IF fbFixClprUnclampChk.udiStatus = 1504 OR fbRmtClprUnclampChk.udiStatus = 1504 THEN
								udiStatus	:= 10002;	//Clamper Clamp Sensor Off Time Out In Unclamp Check While Conveyor Initial With Clamper
							ELSIF fbFixClprUnclampChk.udiStatus = 1505 OR fbRmtClprUnclampChk.udiStatus = 1505 THEN
								udiStatus	:= 10003;	//Clamper Unclamp Sensor On Time Out In Unclamp Check While Conveyor Initial With Clamper
							ELSIF fbFixClprUnclampChk.udiStatus = 1508 OR fbRmtClprUnclampChk.udiStatus = 1508 THEN
								udiStatus	:= 10004;	//Clamper Unclamp Safety Sensor Error In Unclamp Check While Conveyor Initial With Clamper
							ELSE
								IF fbFixClprUnclampChk.udiStatus > 0 AND fbFixClprUnclampChk.udiStatus < 65534 THEN
									udiStatus	:= fbFixClprUnclampChk.udiStatus;
								ELSIF fbRmtClprUnclampChk.udiStatus > 0 AND fbRmtClprUnclampChk.udiStatus < 65534 THEN
									udiStatus	:= fbRmtClprUnclampChk.udiStatus;
								END_IF
							END_IF
						END_IF

					1:	//Magazine Conveyor Init Run
						//Detect Have Magazine
						IF p_bLeftSen OR p_bRightSen THEN
							bHvMag	:= TRUE;
						ELSE
							bHvMag	:= FALSE;
						END_IF

						fbInit.bConvLToR	:= (p_eDirection = ConvDirLToR) OR (p_eDirection = ConvDirLToL);
						fbInit.tTxDlyTm		:= DINT_TO_TIME(p_diInitTm);

						IF fbInit.bConvLToR = TRUE THEN
							fbInit.bEndSen	:= p_bRightSen;
						ELSE
							fbInit.bEndSen	:= p_bLeftSen;
						END_IF

						fbInit(bEn := TRUE);

						bMtrSigOnOrLToR	:= fbInit.bMtrSigOnOrLToR;
						bMtrDirOrRToL	:= fbInit.bMtrDirOrRToL;

						IF fbInit.udiStatus = 0 THEN
							IF fbInit.bConvLToR = TRUE THEN
								IF bHvMag = TRUE AND p_bRightSen = FALSE THEN
									udiStatus	:= 10005;	//Magazine Detected But Not Present At Outlet Sensor (L - R) While Conveyor Initial With Clamper
									eStatus		:= Error;
								ELSE
									usiStep	:= 2;
								END_IF
							ELSE
								IF bHvMag = TRUE AND p_bLeftSen = FALSE THEN
									udiStatus	:= 10006;	//Magazine Detected But Not Present At Outlet Sensor (R - L) While Conveyor Initial With Clamper
									eStatus		:= Error;
								ELSE
									usiStep	:= 2;
								END_IF
							END_IF
						ELSIF fbInit.udiStatus < 65534 THEN
							udiStatus	:= fbInit.udiStatus;
							eStatus		:= Error;
						END_IF

					2:	//Check If Have Magazine
						IF bHvMag = TRUE THEN
							fbWidthChk(IN := NOT p_bWidthChkInterrupt);
							IF p_bWidthChkInterrupt = FALSE THEN
								IF fbWidthChk.Q THEN
									udiStatus := 10048;
									eStatus	  := Error; //Safety Sensor Is Deactivated Before Clamp
								END_IF
							ELSIF p_bWidthChkInterrupt THEN
								usiStep	  := 3;
							END_IF
						ELSE
							eStatus	:= Done;
						END_IF

					3:	//Fix Clamp
						bFixClprClampCtrl	:= TRUE;

						fbFixClprClampChk.bExtSen		:= p_bFixClprClampSen;
						fbFixClprClampChk.bRetSen		:= p_bFixClprUnclampSen;
						fbFixClprClampChk.bExtSafety	:= p_bFixClprClampSafetySen;
						fbFixClprClampChk(bEn := TRUE);

						IF fbFixClprClampChk.udiStatus = 0 THEN
								fbFixClprDly (IN := TRUE);
							IF  fbFixClprDly.Q THEN
								fbFixClprDly (IN := FALSE);
								usiStep	:= 4;
							END_IF

						ELSIF fbFixClprClampChk.udiStatus < 65534 THEN
							bFixClprClampCtrl	:= FALSE;

							eStatus	:= Error;

							IF fbFixClprClampChk.udiStatus = 1503 THEN
								udiStatus	:= 10007;	//Clamper Clamp Sensor On Time Out In Clamp Check While Conveyor Initial With Clamper
							ELSIF fbFixClprClampChk.udiStatus = 1506 THEN
								udiStatus	:= 10008;	//Clamper Unclamp Sensor Off Time Out In Clamp Check While Conveyor Initial With Clamper
							ELSIF fbFixClprClampChk.udiStatus = 1507 THEN
								udiStatus	:= 10009;	//Clamper Clamp Safety Sensor Error In Clamp Check While Conveyor Initial With Clamper
							ELSE
								udiStatus	:= fbFixClprClampChk.udiStatus;
							END_IF
						END_IF

					4:	//Remote Clamp
						bRmtClprClampCtrl	:= TRUE;

						fbRmtClprClampChk.bExtSen		:= p_bRmtClprClampSen;
						fbRmtClprClampChk.bRetSen		:= p_bRmtClprUnclampSen;
						fbRmtClprClampChk.bExtSafety	:= p_bRmtClprClampSafetySen;
						fbRmtClprClampChk(bEn := TRUE);

						IF fbRmtClprClampChk.udiStatus = 0 THEN
								eStatus	:= Done;

						ELSIF fbRmtClprClampChk.udiStatus < 65534 THEN
							bRmtClprClampCtrl	:= FALSE;

							eStatus	:= Error;

							IF fbRmtClprClampChk.udiStatus = 1503 THEN
								udiStatus	:= 10007;	//Clamper Clamp Sensor On Time Out In Clamp Check While Conveyor Initial With Clamper
							ELSIF fbRmtClprClampChk.udiStatus = 1506 THEN
								udiStatus	:= 10008;	//Clamper Unclamp Sensor Off Time Out In Clamp Check While Conveyor Initial With Clamper
							ELSIF fbRmtClprClampChk.udiStatus = 1507 THEN
								udiStatus	:= 10009;	//Clamper Clamp Safety Sensor Error In Clamp Check While Conveyor Initial With Clamper
							ELSE
								udiStatus	:= fbRmtClprClampChk.udiStatus;
							END_IF
						END_IF

				END_CASE
			END_IF

		MagConv2ClpActInitClpStop:
			IF eStatus = Idle OR eStatus = Busy THEN

				eStatus	:= Busy;

				CASE usiStep OF
					0:	//Unclamp
						bFixClprClampCtrl	:= FALSE;
						bRmtClprClampCtrl	:= FALSE;

						fbFixClprUnclampChk.bExtSen		:= p_bFixClprClampSen;
						fbFixClprUnclampChk.bRetSen		:= p_bFixClprUnclampSen;
						fbFixClprUnclampChk.bRetSafety	:= p_bFixClprUnclampSafetySen;
						fbFixClprUnclampChk(bEn := TRUE);

						fbRmtClprUnclampChk.bExtSen		:= p_bRmtClprClampSen;
						fbRmtClprUnclampChk.bRetSen		:= p_bRmtClprUnclampSen;
						fbRmtClprUnclampChk.bRetSafety	:= p_bRmtClprUnclampSafetySen;
						fbRmtClprUnclampChk(bEn := TRUE);

						IF fbFixClprUnclampChk.udiStatus = 0 AND fbRmtClprUnclampChk.udiStatus = 0 THEN
							usiStep	:= 1;
						ELSIF (fbFixClprUnclampChk.udiStatus > 0 AND fbFixClprUnclampChk.udiStatus < 65534) OR (fbRmtClprUnclampChk.udiStatus > 0 AND fbRmtClprUnclampChk.udiStatus < 65534) THEN
							bFixClprClampCtrl	:= TRUE;
							bRmtClprClampCtrl	:= TRUE;

							eStatus	:= Error;

							IF fbFixClprUnclampChk.udiStatus = 1504 OR fbRmtClprUnclampChk.udiStatus = 1504 THEN
								udiStatus	:= 10002;	//Clamper Clamp Sensor Off Time Out In Unclamp Check While Conveyor Initial With Clamper
							ELSIF fbFixClprUnclampChk.udiStatus = 1505 OR fbRmtClprUnclampChk.udiStatus = 1505 THEN
								udiStatus	:= 10003;	//Clamper Unclamp Sensor On Time Out In Unclamp Check While Conveyor Initial With Clamper
							ELSIF fbFixClprUnclampChk.udiStatus = 1508 OR fbRmtClprUnclampChk.udiStatus = 1508 THEN
								udiStatus	:= 10004;	//Clamper Unclamp Safety Sensor Error In Unclamp Check While Conveyor Initial With Clamper
							ELSE
								IF fbFixClprUnclampChk.udiStatus > 0 AND fbFixClprUnclampChk.udiStatus < 65534 THEN
									udiStatus	:= fbFixClprUnclampChk.udiStatus;
								ELSIF fbRmtClprUnclampChk.udiStatus > 0 AND fbRmtClprUnclampChk.udiStatus < 65534 THEN
									udiStatus	:= fbRmtClprUnclampChk.udiStatus;
								END_IF
							END_IF
						END_IF

					1:	//Magazine Conveyor Init Run & Clamp
						//Detect Have Magazine
						IF p_bLeftSen OR p_bRightSen THEN
							bHvMag	:= TRUE;
						ELSE
							bHvMag	:= FALSE;
						END_IF

						fbInit.bConvLToR	:= (p_eDirection = ConvDirLToR) OR (p_eDirection = ConvDirLToL);
						fbInit.tTxDlyTm		:= DINT_TO_TIME(p_diInitTm);

						IF fbInit.bConvLToR = TRUE THEN
							fbInit.bEndSen	:= p_bRightSen;
						ELSE
							fbInit.bEndSen	:= p_bLeftSen;
						END_IF

						fbInit(bEn := TRUE);

						bMtrSigOnOrLToR	:= fbInit.bMtrSigOnOrLToR;
						bMtrDirOrRToL	:= fbInit.bMtrDirOrRToL;

						IF fbInit.bEndSen = TRUE THEN
							bReachEnd	:= TRUE;
						END_IF

						IF bReachEnd = TRUE THEN
							fbClprDlyTm(IN := TRUE);
							IF fbClprDlyTm.Q = TRUE THEN
								CASE usiSubStep OF
								//	0:	//Fix Clamp
//										bFixClprClampCtrl	:= TRUE;

//										fbFixClprClampChk.bExtSen		:= p_bFixClprClampSen;
//										fbFixClprClampChk.bRetSen		:= p_bFixClprUnclampSen;
//										fbFixClprClampChk.bExtSafety	:= p_bFixClprClampSafetySen;
//										fbFixClprClampChk(bEn := TRUE);
//
//										IF fbFixClprClampChk.udiStatus = 0 THEN
//											usiSubStep	:= 1;
//										END_IF

									0:	//Remote Clamp
										bRmtClprClampCtrl	:= TRUE;

										fbRmtClprClampChk.bExtSen		:= p_bRmtClprClampSen;
										fbRmtClprClampChk.bRetSen		:= p_bRmtClprUnclampSen;
										fbRmtClprClampChk.bExtSafety	:= p_bRmtClprClampSafetySen;
										fbRmtClprClampChk(bEn := TRUE);

										IF fbRmtClprClampChk.udiStatus = 0 THEN
											usiSubStep	:= 1;
										END_IF

									1:

										bFixClprClampCtrl	:= TRUE;

										fbFixClprClampChk.bExtSen		:= p_bFixClprClampSen;
										fbFixClprClampChk.bRetSen		:= p_bFixClprUnclampSen;
										fbFixClprClampChk.bExtSafety	:= p_bFixClprClampSafetySen;
										fbFixClprClampChk(bEn := TRUE);

								END_CASE
							END_IF
						END_IF

						IF (fbInit.udiStatus = 0) AND ((fbFixClprClampChk.udiStatus = 0 AND fbRmtClprClampChk.udiStatus = 0) OR (bReachEnd = FALSE)) THEN
							IF fbInit.bConvLToR = TRUE THEN
								IF bHvMag = TRUE AND p_bRightSen = FALSE THEN
									udiStatus	:= 10041;	//Magazine Detected But Not Present At Outlet Sensor (L - R) While Conveyor Initial With Clamper
									eStatus		:= Error;
								ELSE
									eStatus		:= Done;
								END_IF
							ELSE
								IF bHvMag = TRUE AND p_bLeftSen = FALSE THEN
									udiStatus	:= 10042;	//Magazine Detected But Not Present At Outlet Sensor (R - L) While Conveyor Initial With Clamper
									eStatus		:= Error;
								ELSE
									eStatus		:= Done;
								END_IF
							END_IF

						ELSIF fbInit.udiStatus > 0 AND fbInit.udiStatus < 65534 THEN
							udiStatus	:= fbInit.udiStatus;
							eStatus		:= Error;

						ELSIF (fbFixClprClampChk.udiStatus > 0 AND fbFixClprClampChk.udiStatus < 65534) OR (fbRmtClprClampChk.udiStatus > 0 AND fbRmtClprClampChk.udiStatus < 65534) THEN
							bFixClprClampCtrl	:= FALSE;
							bRmtClprClampCtrl	:= FALSE;

							eStatus	:= Error;

							IF fbFixClprClampChk.udiStatus = 1503 OR fbRmtClprClampChk.udiStatus = 1503 THEN
								udiStatus	:= 10043;	//Clamper Clamp Sensor On Time Out In Clamp Check While Conveyor Initial With Clamper
							ELSIF fbFixClprClampChk.udiStatus = 1506 OR fbRmtClprClampChk.udiStatus = 1506 THEN
								udiStatus	:= 10044;	//Clamper Unclamp Sensor Off Time Out In Clamp Check While Conveyor Initial With Clamper
							ELSIF fbFixClprClampChk.udiStatus = 1507 OR fbRmtClprClampChk.udiStatus = 1507 THEN
								udiStatus	:= 10045;	//Clamper Clamp Safety Sensor Error In Clamp Check While Conveyor Initial With Clamper
							ELSE
								IF fbFixClprClampChk.udiStatus > 0 AND fbFixClprClampChk.udiStatus < 65534 THEN
									udiStatus	:= fbFixClprClampChk.udiStatus;
								ELSIF fbRmtClprClampChk.udiStatus > 0 AND fbRmtClprClampChk.udiStatus < 65534 THEN
									udiStatus	:= fbRmtClprClampChk.udiStatus;
								END_IF
							END_IF
						END_IF

				END_CASE
			END_IF

		MagConv2ClpActEnt:
			IF eStatus = Idle OR eStatus = Busy THEN

				eStatus	:= Busy;

				//Detect Have Magazine
				IF p_bLeftSen OR p_bRightSen THEN
					bHvMag	:= TRUE;
				END_IF

				//Conveyor Run
				fbEnt.bConvLToR		:= (p_eDirection = ConvDirLToR) OR (p_eDirection = ConvDirLToL);
				fbEnt.tTimeOut		:= DINT_TO_TIME(p_diTxInTimeOut);

				IF fbEnt.bConvLToR = TRUE THEN
					fbEnt.bEndSen	:= p_bRightSen;
				ELSE
					fbEnt.bEndSen	:= p_bLeftSen;
				END_IF

				fbEnt(bEn := TRUE);

				bMtrSigOnOrLToR	:= fbEnt.bMtrSigOnOrLToR;
				bMtrDirOrRToL	:= fbEnt.bMtrDirOrRToL;

				IF fbEnt.udiStatus = 0 THEN
					eStatus		:= Done;
				ELSIF fbEnt.udiStatus < 65534 THEN
					eStatus		:= Error;

					IF fbEnt.udiStatus = 1101 THEN
						udiStatus	:= 10028;	//Transfer In Time Out While Entering Magazine
					ELSE
						udiStatus	:= fbEnt.udiStatus;
					END_IF
				END_IF

			END_IF

		MagConv2ClpActEntStopClp:
			IF eStatus = Idle OR eStatus = Busy THEN

				eStatus	:= Busy;

				CASE usiStep OF
					0:	//Conveyor Enter
						//Detect Have Magazine
						IF p_bLeftSen OR p_bRightSen THEN
							bHvMag	:= TRUE;
						END_IF

						//Conveyor Run
						fbEnt.bConvLToR		:= (p_eDirection = ConvDirLToR) OR (p_eDirection = ConvDirLToL);
						fbEnt.tTimeOut		:= DINT_TO_TIME(p_diTxInTimeOut);

						IF fbEnt.bConvLToR = TRUE THEN
							fbEnt.bEndSen	:= p_bRightSen;
						ELSE
							fbEnt.bEndSen	:= p_bLeftSen;
						END_IF

						fbEnt(bEn := TRUE);

						bMtrSigOnOrLToR	:= fbEnt.bMtrSigOnOrLToR;
						bMtrDirOrRToL	:= fbEnt.bMtrDirOrRToL;

						IF fbEnt.udiStatus = 0 THEN
//							usiStep	:= 1;
							fbWidthChk(IN := NOT p_bWidthChkInterrupt);
								IF p_bWidthChkInterrupt = FALSE THEN
								    IF fbWidthChk.Q THEN
										udiStatus := 10048;
										eStatus	  := Error; //Safety Sensor Is Deactivated Before Clamp
									END_IF
								ELSIF p_bWidthChkInterrupt THEN
									usiStep	  := 1;
								END_IF
						ELSIF fbEnt.udiStatus < 65534 THEN
							eStatus	:= Error;

							IF fbEnt.udiStatus = 1101 THEN
								udiStatus	:= 10029;	//Transfer In Time Out While Entering Magazine
							ELSE
								udiStatus	:= fbEnt.udiStatus;
							END_IF
						END_IF

					1:	//Fix Clamp
						bFixClprClampCtrl	:= TRUE;

						fbFixClprClampChk.bExtSen		:= p_bFixClprClampSen;
						fbFixClprClampChk.bRetSen		:= p_bFixClprUnclampSen;
						fbFixClprClampChk.bExtSafety	:= p_bFixClprClampSafetySen;
						fbFixClprClampChk(bEn := TRUE);

						IF fbFixClprClampChk.udiStatus = 0 THEN
							fbFixClprDly(IN := TRUE);
							IF  fbFixClprDly.Q THEN
								fbFixClprDly (IN := FALSE);
								usiStep	:= 2;
							END_IF

						ELSIF fbFixClprClampChk.udiStatus < 65534 THEN
							bFixClprClampCtrl	:= FALSE;

							eStatus	:= Error;

							IF fbFixClprClampChk.udiStatus = 1503 THEN
								udiStatus	:= 10010;	//Clamper Clamp Sensor On Time Out In Clamp Check While Conveyor Enter With Clamper
							ELSIF fbFixClprClampChk.udiStatus = 1506 THEN
								udiStatus	:= 10011;	//Clamper Unclamp Sensor Off Time Out In Clamp Check While Conveyor Enter With Clamper
							ELSIF fbFixClprClampChk.udiStatus = 1507 THEN
								udiStatus	:= 10012;	//Clamper Clamp Safety Sensor Error In Clamp Check While Conveyor Enter With Clamper
							ELSE
								udiStatus	:= fbFixClprClampChk.udiStatus;
							END_IF
						END_IF

					2:	//Remote Clamp
						bRmtClprClampCtrl	:= TRUE;

						fbRmtClprClampChk.bExtSen		:= p_bRmtClprClampSen;
						fbRmtClprClampChk.bRetSen		:= p_bRmtClprUnclampSen;
						fbRmtClprClampChk.bExtSafety	:= p_bRmtClprClampSafetySen;
						fbRmtClprClampChk(bEn := TRUE);

						IF fbRmtClprClampChk.udiStatus = 0 THEN
								eStatus	:= Done;

						ELSIF fbRmtClprClampChk.udiStatus < 65534 THEN
							bRmtClprClampCtrl	:= FALSE;

							eStatus	:= Error;

							IF fbRmtClprClampChk.udiStatus = 1503 THEN
								udiStatus	:= 10010;	//Clamper Clamp Sensor On Time Out In Clamp Check While Conveyor Enter With Clamper
							ELSIF fbRmtClprClampChk.udiStatus = 1506 THEN
								udiStatus	:= 10011;	//Clamper Unclamp Sensor Off Time Out In Clamp Check While Conveyor Enter With Clamper
							ELSIF fbRmtClprClampChk.udiStatus = 1507 THEN
								udiStatus	:= 10012;	//Clamper Clamp Safety Sensor Error In Clamp Check While Conveyor Enter With Clamper
							ELSE
								udiStatus	:= fbRmtClprClampChk.udiStatus;
							END_IF
						END_IF

				END_CASE

			END_IF

		MagConv2ClpActEntClpStop:
			IF eStatus = Idle OR eStatus = Busy THEN

				eStatus	:= Busy;

				//Detect Have Magazine
				IF p_bLeftSen OR p_bRightSen THEN
					bHvMag	:= TRUE;
				END_IF

				//Conveyor Run
				fbEnt.bConvLToR		:= (p_eDirection = ConvDirLToR) OR (p_eDirection = ConvDirLToL);
				fbEnt.tTimeOut		:= DINT_TO_TIME(p_diTxInTimeOut);

				IF fbEnt.bConvLToR = TRUE THEN
					fbEnt.bEndSen	:= p_bRightSen;
				ELSE
					fbEnt.bEndSen	:= p_bLeftSen;
				END_IF

				fbEnt(bEn := TRUE);

				bMtrSigOnOrLToR	:= fbEnt.bMtrSigOnOrLToR;
				bMtrDirOrRToL	:= fbEnt.bMtrDirOrRToL;

				IF fbEnt.bEndSen = TRUE THEN
					bReachEnd	:= TRUE;
				END_IF

				IF bReachEnd = TRUE THEN
					fbClprDlyTm(IN := TRUE);
					IF fbClprDlyTm.Q = TRUE THEN
						CASE usiSubStep OF
							0:	//Fix Clamp
//								bFixClprClampCtrl	:= TRUE;
//
//								fbFixClprClampChk.bExtSen		:= p_bFixClprClampSen;
//								fbFixClprClampChk.bRetSen		:= p_bFixClprUnclampSen;
//								fbFixClprClampChk.bExtSafety	:= p_bFixClprClampSafetySen;
//								fbFixClprClampChk(bEn := TRUE);
//
//								IF fbFixClprClampChk.udiStatus = 0 THEN
//									usiSubStep	:= 1;
//								END_IF

								bRmtClprClampCtrl	:= TRUE;

								fbRmtClprClampChk.bExtSen		:= p_bRmtClprClampSen;
								fbRmtClprClampChk.bRetSen		:= p_bRmtClprUnclampSen;
								fbRmtClprClampChk.bExtSafety	:= p_bRmtClprClampSafetySen;
								fbRmtClprClampChk(bEn := TRUE);

								IF fbRmtClprClampChk.udiStatus = 0 THEN
									usiSubStep	:= 1;
								END_IF

							1:	//Remote Clamp
//								bRmtClprClampCtrl	:= TRUE;
//
//								fbRmtClprClampChk.bExtSen		:= p_bRmtClprClampSen;
//								fbRmtClprClampChk.bRetSen		:= p_bRmtClprUnclampSen;
//								fbRmtClprClampChk.bExtSafety	:= p_bRmtClprClampSafetySen;
//								fbRmtClprClampChk(bEn := TRUE);

								bFixClprClampCtrl	:= TRUE;

								fbFixClprClampChk.bExtSen		:= p_bFixClprClampSen;
								fbFixClprClampChk.bRetSen		:= p_bFixClprUnclampSen;
								fbFixClprClampChk.bExtSafety	:= p_bFixClprClampSafetySen;
								fbFixClprClampChk(bEn := TRUE);

						END_CASE
					END_IF
				END_IF

				IF fbEnt.udiStatus = 0 AND (fbFixClprClampChk.udiStatus = 0 AND fbRmtClprClampChk.udiStatus = 0) THEN
					eStatus	:= Done;

				ELSIF (fbFixClprClampChk.udiStatus > 0 AND fbFixClprClampChk.udiStatus < 65534) OR (fbRmtClprClampChk.udiStatus > 0 AND fbRmtClprClampChk.udiStatus < 65534) THEN
					bFixClprClampCtrl	:= FALSE;
					bRmtClprClampCtrl	:= FALSE;

					eStatus	:= Error;

					IF fbFixClprClampChk.udiStatus = 1503 OR fbRmtClprClampChk.udiStatus = 1503 THEN
						udiStatus	:= 10034;	//Clamper Clamp Sensor On Time Out In Clamp Check While Conveyor Enter With Clamper
					ELSIF fbFixClprClampChk.udiStatus = 1506 OR fbRmtClprClampChk.udiStatus = 1506 THEN
						udiStatus	:= 10035;	//Clamper Unclamp Sensor Off Time Out In Clamp Check While Conveyor Enter With Clamper
					ELSIF fbFixClprClampChk.udiStatus = 1507 OR fbRmtClprClampChk.udiStatus = 1507 THEN
						udiStatus	:= 10036;	//Clamper Clamp Safety Sensor Error In Clamp Check While Conveyor Enter With Clamper
					ELSE
						IF fbFixClprClampChk.udiStatus > 0 AND fbFixClprClampChk.udiStatus < 65534 THEN
							udiStatus	:= fbFixClprClampChk.udiStatus;
						ELSIF fbRmtClprClampChk.udiStatus > 0 AND fbRmtClprClampChk.udiStatus < 65534 THEN
							udiStatus	:= fbRmtClprClampChk.udiStatus;
						END_IF
					END_IF

				ELSIF fbEnt.udiStatus > 0 AND fbEnt.udiStatus < 65534 THEN
					eStatus	:= Error;

					IF fbEnt.udiStatus = 1101 THEN
						udiStatus	:= 10037;	//Transfer In Time Out While Entering Magazine
					ELSE
						udiStatus	:= fbEnt.udiStatus;
					END_IF

				END_IF

			END_IF

		MagConv2ClpActPreExit:
			IF eStatus = Idle OR eStatus = Busy THEN

				eStatus	:= Busy;

				//Conveyor Run
				fbPreExit.bConvLToR		:= (p_eDirection = ConvDirLToR) OR (p_eDirection = ConvDirRToR);
				fbPreExit.tTxDlyTm		:= DINT_TO_TIME(p_diInitTm);

				IF fbPreExit.bConvLToR = TRUE THEN
					fbPreExit.bEndSen	:= p_bRightSen;
					fbPreExit.bStartSen	:= p_bLeftSen;
				ELSE
					fbPreExit.bEndSen	:= p_bLeftSen;
					fbPreExit.bStartSen	:= p_bRightSen;
				END_IF

				fbPreExit(bEn := TRUE);

				bMtrSigOnOrLToR	:= fbPreExit.bMtrSigOnOrLToR;
				bMtrDirOrRToL	:= fbPreExit.bMtrDirOrRToL;

				IF fbPreExit.udiStatus = 0 THEN
					IF fbPreExit.bEndSen = TRUE THEN
						eStatus	:= Done;
					ELSE
						udiStatus	:= 10046;	//Magazine Not Detected While Pre-Exiting Magazine
						eStatus		:= Error;
					END_IF
				ELSIF fbPreExit.udiStatus < 65534 THEN
					udiStatus	:= fbPreExit.udiStatus;
					eStatus		:= Error;
				END_IF

			END_IF

		MagConv2ClpActPreExitClpr:
			IF eStatus = Idle OR eStatus = Busy THEN

				eStatus	:= Busy;

				CASE usiStep OF
					0:	//Unclamp
						bFixClprClampCtrl	:= FALSE;
						bRmtClprClampCtrl	:= FALSE;

						fbFixClprUnclampChk.bExtSen		:= p_bFixClprClampSen;
						fbFixClprUnclampChk.bRetSen		:= p_bFixClprUnclampSen;
						fbFixClprUnclampChk.bRetSafety	:= p_bFixClprUnclampSafetySen;
						fbFixClprUnclampChk(bEn := TRUE);

						fbRmtClprUnclampChk.bExtSen		:= p_bRmtClprClampSen;
						fbRmtClprUnclampChk.bRetSen		:= p_bRmtClprUnclampSen;
						fbRmtClprUnclampChk.bRetSafety	:= p_bRmtClprUnclampSafetySen;
						fbRmtClprUnclampChk(bEn := TRUE);

						IF fbFixClprUnclampChk.udiStatus = 0 AND fbRmtClprUnclampChk.udiStatus = 0 THEN
							usiStep	:= 1;
						ELSIF (fbFixClprUnclampChk.udiStatus > 0 AND fbFixClprUnclampChk.udiStatus < 65534) OR (fbRmtClprUnclampChk.udiStatus > 0 AND fbRmtClprUnclampChk.udiStatus < 65534) THEN
							bFixClprClampCtrl	:= TRUE;
							bRmtClprClampCtrl	:= TRUE;

							eStatus	:= Error;

							IF fbFixClprUnclampChk.udiStatus = 1504 OR fbRmtClprUnclampChk.udiStatus = 1504 THEN
								udiStatus	:= 10002;	//Clamper Clamp Sensor Off Time Out In Unclamp Check While Conveyor Initial With Clamper
							ELSIF fbFixClprUnclampChk.udiStatus = 1505 OR fbRmtClprUnclampChk.udiStatus = 1505 THEN
								udiStatus	:= 10003;	//Clamper Unclamp Sensor On Time Out In Unclamp Check While Conveyor Initial With Clamper
							ELSIF fbFixClprUnclampChk.udiStatus = 1508 OR fbRmtClprUnclampChk.udiStatus = 1508 THEN
								udiStatus	:= 10004;	//Clamper Unclamp Safety Sensor Error In Unclamp Check While Conveyor Initial With Clamper
							ELSE
								IF fbFixClprUnclampChk.udiStatus > 0 AND fbFixClprUnclampChk.udiStatus < 65534 THEN
									udiStatus	:= fbFixClprUnclampChk.udiStatus;
								ELSIF fbRmtClprUnclampChk.udiStatus > 0 AND fbRmtClprUnclampChk.udiStatus < 65534 THEN
									udiStatus	:= fbRmtClprUnclampChk.udiStatus;
								END_IF
							END_IF
						END_IF

					1:	//Conveyor Pre-Exit
						//Conveyor Run
						fbPreExit.bConvLToR		:= (p_eDirection = ConvDirLToR) OR (p_eDirection = ConvDirRToR);
						fbPreExit.tTxDlyTm		:= DINT_TO_TIME(p_diInitTm);

						IF fbPreExit.bConvLToR = TRUE THEN
							fbPreExit.bEndSen	:= p_bRightSen;
							fbPreExit.bStartSen	:= p_bLeftSen;
						ELSE
							fbPreExit.bEndSen	:= p_bLeftSen;
							fbPreExit.bStartSen	:= p_bRightSen;
						END_IF

						fbPreExit(bEn := TRUE);

						bMtrSigOnOrLToR	:= fbPreExit.bMtrSigOnOrLToR;
						bMtrDirOrRToL	:= fbPreExit.bMtrDirOrRToL;

						IF fbPreExit.udiStatus = 0 THEN
							IF fbPreExit.bEndSen = TRUE THEN
								eStatus	:= Done;
							ELSE
								udiStatus	:= 10046;	//Magazine Not Detected While Pre-Exiting Magazine
								eStatus		:= Error;
							END_IF
						ELSIF fbPreExit.udiStatus < 65534 THEN
							udiStatus	:= fbPreExit.udiStatus;
							eStatus		:= Error;
						END_IF

				END_CASE

			END_IF

		MagConv2ClpActExit:
			IF eStatus = Idle OR eStatus = Busy THEN

				eStatus	:= Busy;

				//Conveyor Run
				fbExit.bConvLToR	:= (p_eDirection = ConvDirLToR) OR (p_eDirection = ConvDirRToR);
				fbExit.tTimeOut		:= DINT_TO_TIME(p_diTxOutTimeOut);

				IF fbExit.bConvLToR = TRUE THEN
					fbExit.bEndSen	:= p_bRightSen;
				ELSE
					fbExit.bEndSen	:= p_bLeftSen;
				END_IF

				fbExit(bEn := TRUE);

				bMtrSigOnOrLToR	:= fbExit.bMtrSigOnOrLToR;
				bMtrDirOrRToL	:= fbExit.bMtrDirOrRToL;

				IF fbExit.udiStatus = 0 THEN
					bHvMag		:= FALSE;
					eStatus		:= Done;
				ELSIF fbExit.udiStatus < 65534 THEN
					eStatus		:= Error;

					IF fbExit.udiStatus = 1101 THEN
						udiStatus	:= 10030;	//Transfer Out Time Out While Exiting Magazine
					ELSE
						udiStatus	:= fbExit.udiStatus;
					END_IF
				END_IF

			END_IF

		MagConv2ClpActExit1:
			IF eStatus = Idle OR eStatus = Busy THEN

				eStatus	:= Busy;

				//Conveyor Run
				fbExit1.bConvLToR		:= (p_eDirection = ConvDirLToR) OR (p_eDirection = ConvDirRToR);
				fbExit1.tTimeOut		:= DINT_TO_TIME(p_diTxOutTimeOut);

				IF fbExit1.bConvLToR = TRUE THEN
					fbExit1.bEndSen	:= p_bRightSen;
				ELSE
					fbExit1.bEndSen	:= p_bLeftSen;
				END_IF

				fbExit1(bEn := TRUE);

				bMtrSigOnOrLToR	:= fbExit1.bMtrSigOnOrLToR;
				bMtrDirOrRToL	:= fbExit1.bMtrDirOrRToL;

				IF fbExit1.udiStatus = 0 THEN
					bHvMag		:= FALSE;
					eStatus		:= Done;
				ELSIF fbExit1.udiStatus < 65534 THEN
					eStatus		:= Error;

					IF fbExit1.udiStatus = 1101 THEN
						udiStatus	:= 10032;	//Transfer Out Time Out While Exiting Magazinie
					ELSE
						udiStatus	:= fbExit1.udiStatus;
					END_IF
				END_IF

			END_IF

		MagConv2ClpActExitClpr:
			IF eStatus = Idle OR eStatus = Busy THEN

				eStatus	:= Busy;

				CASE usiStep OF
					0:	//Unclamp
						bFixClprClampCtrl	:= FALSE;
						bRmtClprClampCtrl	:= FALSE;

						fbFixClprUnclampChk.bExtSen		:= p_bFixClprClampSen;
						fbFixClprUnclampChk.bRetSen		:= p_bFixClprUnclampSen;
						fbFixClprUnclampChk.bRetSafety	:= p_bFixClprUnclampSafetySen;
						fbFixClprUnclampChk(bEn := TRUE);

						fbRmtClprUnclampChk.bExtSen		:= p_bRmtClprClampSen;
						fbRmtClprUnclampChk.bRetSen		:= p_bRmtClprUnclampSen;
						fbRmtClprUnclampChk.bRetSafety	:= p_bRmtClprUnclampSafetySen;
						fbRmtClprUnclampChk(bEn := TRUE);

						IF fbFixClprUnclampChk.udiStatus = 0 AND fbRmtClprUnclampChk.udiStatus = 0 THEN
							usiStep	:= 1;
						ELSIF (fbFixClprUnclampChk.udiStatus > 0 AND fbFixClprUnclampChk.udiStatus < 65534) OR (fbRmtClprUnclampChk.udiStatus > 0 AND fbRmtClprUnclampChk.udiStatus < 65534) THEN
							bFixClprClampCtrl	:= TRUE;
							bRmtClprClampCtrl	:= TRUE;

							eStatus	:= Error;

							IF fbFixClprUnclampChk.udiStatus = 1504 OR fbRmtClprUnclampChk.udiStatus = 1504 THEN
								udiStatus	:= 10002;	//Clamper Clamp Sensor Off Time Out In Unclamp Check While Conveyor Initial With Clamper
							ELSIF fbFixClprUnclampChk.udiStatus = 1505 OR fbRmtClprUnclampChk.udiStatus = 1505 THEN
								udiStatus	:= 10003;	//Clamper Unclamp Sensor On Time Out In Unclamp Check While Conveyor Initial With Clamper
							ELSIF fbFixClprUnclampChk.udiStatus = 1508 OR fbRmtClprUnclampChk.udiStatus = 1508 THEN
								udiStatus	:= 10004;	//Clamper Unclamp Safety Sensor Error In Unclamp Check While Conveyor Initial With Clamper
							ELSE
								IF fbFixClprUnclampChk.udiStatus > 0 AND fbFixClprUnclampChk.udiStatus < 65534 THEN
									udiStatus	:= fbFixClprUnclampChk.udiStatus;
								ELSIF fbRmtClprUnclampChk.udiStatus > 0 AND fbRmtClprUnclampChk.udiStatus < 65534 THEN
									udiStatus	:= fbRmtClprUnclampChk.udiStatus;
								END_IF
							END_IF
						END_IF

					1:	//Conveyor Exit
						//Conveyor Run
						fbExit.bConvLToR	:= (p_eDirection = ConvDirLToR) OR (p_eDirection = ConvDirRToR);
						fbExit.tTimeOut		:= DINT_TO_TIME(p_diTxOutTimeOut);

						IF fbExit.bConvLToR = TRUE THEN
							fbExit.bEndSen	:= p_bRightSen;
						ELSE
							fbExit.bEndSen	:= p_bLeftSen;
						END_IF

						fbExit(bEn := TRUE);

						bMtrSigOnOrLToR	:= fbExit.bMtrSigOnOrLToR;
						bMtrDirOrRToL	:= fbExit.bMtrDirOrRToL;

						IF fbExit.udiStatus = 0 THEN
							bHvMag		:= FALSE;
							eStatus		:= Done;
						ELSIF fbExit.udiStatus < 65534 THEN
							eStatus		:= Error;

							IF fbExit.udiStatus = 1101 THEN
								udiStatus	:= 10031;	//Transfer Out Time Out While Conveyor Exit With Clamper
							ELSE
								udiStatus	:= fbExit.udiStatus;
							END_IF
						END_IF

				END_CASE

			END_IF

		MagConv2ClpActExit1Clpr:
			IF eStatus = Idle OR eStatus = Busy THEN

				eStatus	:= Busy;

				CASE usiStep OF
					0:	//Unclamp
						bFixClprClampCtrl	:= FALSE;
						bRmtClprClampCtrl	:= FALSE;

						fbFixClprUnclampChk.bExtSen		:= p_bFixClprClampSen;
						fbFixClprUnclampChk.bRetSen		:= p_bFixClprUnclampSen;
						fbFixClprUnclampChk.bRetSafety	:= p_bFixClprUnclampSafetySen;
						fbFixClprUnclampChk(bEn := TRUE);

						fbRmtClprUnclampChk.bExtSen		:= p_bRmtClprClampSen;
						fbRmtClprUnclampChk.bRetSen		:= p_bRmtClprUnclampSen;
						fbRmtClprUnclampChk.bRetSafety	:= p_bRmtClprUnclampSafetySen;
						fbRmtClprUnclampChk(bEn := TRUE);

						IF fbFixClprUnclampChk.udiStatus = 0 AND fbRmtClprUnclampChk.udiStatus = 0 THEN
							usiStep	:= 1;
						ELSIF (fbFixClprUnclampChk.udiStatus > 0 AND fbFixClprUnclampChk.udiStatus < 65534) OR (fbRmtClprUnclampChk.udiStatus > 0 AND fbRmtClprUnclampChk.udiStatus < 65534) THEN
							bFixClprClampCtrl	:= TRUE;
							bRmtClprClampCtrl	:= TRUE;

							eStatus	:= Error;

							IF fbFixClprUnclampChk.udiStatus = 1504 OR fbRmtClprUnclampChk.udiStatus = 1504 THEN
								udiStatus	:= 10002;	//Clamper Clamp Sensor Off Time Out In Unclamp Check While Conveyor Initial With Clamper
							ELSIF fbFixClprUnclampChk.udiStatus = 1505 OR fbRmtClprUnclampChk.udiStatus = 1505 THEN
								udiStatus	:= 10003;	//Clamper Unclamp Sensor On Time Out In Unclamp Check While Conveyor Initial With Clamper
							ELSIF fbFixClprUnclampChk.udiStatus = 1508 OR fbRmtClprUnclampChk.udiStatus = 1508 THEN
								udiStatus	:= 10004;	//Clamper Unclamp Safety Sensor Error In Unclamp Check While Conveyor Initial With Clamper
							ELSE
								IF fbFixClprUnclampChk.udiStatus > 0 AND fbFixClprUnclampChk.udiStatus < 65534 THEN
									udiStatus	:= fbFixClprUnclampChk.udiStatus;
								ELSIF fbRmtClprUnclampChk.udiStatus > 0 AND fbRmtClprUnclampChk.udiStatus < 65534 THEN
									udiStatus	:= fbRmtClprUnclampChk.udiStatus;
								END_IF
							END_IF
						END_IF

					1:	//Conveyor Exit
						//Conveyor Run
						fbExit1.bConvLToR		:= (p_eDirection = ConvDirLToR) OR (p_eDirection = ConvDirRToR);
						fbExit1.tTimeOut		:= DINT_TO_TIME(p_diTxOutTimeOut);

						IF fbExit1.bConvLToR = TRUE THEN
							fbExit1.bEndSen	:= p_bRightSen;
						ELSE
							fbExit1.bEndSen	:= p_bLeftSen;
						END_IF

						fbExit1(bEn := TRUE);

						bMtrSigOnOrLToR	:= fbExit1.bMtrSigOnOrLToR;
						bMtrDirOrRToL	:= fbExit1.bMtrDirOrRToL;

						IF fbExit1.udiStatus = 0 THEN
							bHvMag		:= FALSE;
							eStatus		:= Done;
						ELSIF fbExit1.udiStatus < 65534 THEN
							eStatus		:= Error;

							IF fbExit1.udiStatus = 1101 THEN
								udiStatus	:= 10033;	//Transfer Out Time Out While Conveyor Exit With Clamper
							ELSE
								udiStatus	:= fbExit1.udiStatus;
							END_IF
						END_IF

				END_CASE

			END_IF

		MagConv2ClpActFixClprSetAll:
			IF eStatus = Idle OR eStatus = Busy THEN

				eStatus	:= Busy;

				bMtrSigOnOrLToR	:= FALSE;
				bMtrDirOrRToL	:= FALSE;

				bFixClprClampCtrl	:= TRUE;

				eStatus	:= Done;

			END_IF

		MagConv2ClpActFixClprRstAll:
			IF eStatus = Idle OR eStatus = Busy THEN

				eStatus	:= Busy;

				bMtrSigOnOrLToR	:= FALSE;
				bMtrDirOrRToL	:= FALSE;

				bFixClprClampCtrl	:= FALSE;

				eStatus	:= Done;

			END_IF

		MagConv2ClpActFixClprSetClamp:
			IF eStatus = Idle OR eStatus = Busy THEN

				eStatus	:= Busy;

				bMtrSigOnOrLToR	:= FALSE;
				bMtrDirOrRToL	:= FALSE;

				bFixClprClampCtrl	:= TRUE;

				eStatus	:= Done;

			END_IF

		MagConv2ClpActFixClprSetUnclamp:
			IF eStatus = Idle OR eStatus = Busy THEN

				eStatus	:= Busy;

				bMtrSigOnOrLToR	:= FALSE;
				bMtrDirOrRToL	:= FALSE;

				bFixClprClampCtrl	:= FALSE;

				eStatus	:= Done;

			END_IF

		MagConv2ClpActFixClprClamp:
			IF eStatus = Idle OR eStatus = Busy THEN

				eStatus	:= Busy;

				bMtrSigOnOrLToR	:= FALSE;
				bMtrDirOrRToL	:= FALSE;

				bFixClprClampCtrl	:= TRUE;

				fbFixClprClampChk.bExtSen		:= p_bFixClprClampSen;
				fbFixClprClampChk.bRetSen		:= p_bFixClprUnclampSen;
				fbFixClprClampChk.bExtSafety	:= p_bFixClprClampSafetySen;
				fbFixClprClampChk(bEn := TRUE);

				IF fbFixClprClampChk.udiStatus = 0 THEN
					eStatus	:= Done;
				ELSIF fbFixClprClampChk.udiStatus < 65534 THEN
					bFixClprClampCtrl	:= FALSE;

					eStatus	:= Error;

					IF fbFixClprClampChk.udiStatus = 1503 THEN
						udiStatus	:= 10016;	//Clamper Clamp Sensor On Time Out In Clamp Check While Clamper Clamp
					ELSIF fbFixClprClampChk.udiStatus = 1506 THEN
						udiStatus	:= 10017;	//Clamper Unclamp Sensor Off Time Out In Clamp Check While Clamper Clamp
					ELSIF fbFixClprClampChk.udiStatus = 1507 THEN
						udiStatus	:= 10018;	//Clamper Clamp Safety Sensor Error In Clamp Check While Clamper Clamp
					ELSE
						udiStatus	:= fbFixClprClampChk.udiStatus;
					END_IF
				END_IF
			END_IF

		MagConv2ClpActFixClprUnclamp:
			IF eStatus = Idle OR eStatus = Busy THEN

				eStatus	:= Busy;

				bMtrSigOnOrLToR	:= FALSE;
				bMtrDirOrRToL	:= FALSE;

				bFixClprClampCtrl	:= FALSE;

				fbFixClprUnclampChk.bExtSen		:= p_bFixClprClampSen;
				fbFixClprUnclampChk.bRetSen		:= p_bFixClprUnclampSen;
				fbFixClprUnclampChk.bRetSafety	:= p_bFixClprUnclampSafetySen;
				fbFixClprUnclampChk(bEn := TRUE);

				IF fbFixClprUnclampChk.udiStatus = 0 THEN
					eStatus	:= Done;
				ELSIF fbFixClprUnclampChk.udiStatus < 65534 THEN
					bFixClprClampCtrl	:= TRUE;

					eStatus	:= Error;

					IF fbFixClprUnclampChk.udiStatus = 1504 THEN
						udiStatus	:= 10019;	//Clamper Clamp Sensor Off Time Out In Unclamp Check While Clamper Unclamp
					ELSIF fbFixClprUnclampChk.udiStatus = 1505 THEN
						udiStatus	:= 10020;	//Clamper Unclamp Sensor On Time Out In Unclamp Check While Clamper Unclamp
					ELSIF fbFixClprUnclampChk.udiStatus = 1508 THEN
						udiStatus	:= 10021;	//Clamper Unclamp Safety Sensor Error In Unclamp Check While Clamper Unclamp
					ELSE
						udiStatus	:= fbFixClprUnclampChk.udiStatus;
					END_IF
				END_IF

			END_IF

		MagConv2ClpActRmtClprSetAll:
			IF eStatus = Idle OR eStatus = Busy THEN

				eStatus	:= Busy;

				bMtrSigOnOrLToR	:= FALSE;
				bMtrDirOrRToL	:= FALSE;

				bRmtClprClampCtrl	:= TRUE;

				eStatus	:= Done;

			END_IF

		MagConv2ClpActRmtClprRstAll:
			IF eStatus = Idle OR eStatus = Busy THEN

				eStatus	:= Busy;

				bMtrSigOnOrLToR	:= FALSE;
				bMtrDirOrRToL	:= FALSE;

				bRmtClprClampCtrl	:= FALSE;

				eStatus	:= Done;

			END_IF

		MagConv2ClpActRmtClprSetClamp:
			IF eStatus = Idle OR eStatus = Busy THEN

				eStatus	:= Busy;

				bMtrSigOnOrLToR	:= FALSE;
				bMtrDirOrRToL	:= FALSE;

				bRmtClprClampCtrl	:= TRUE;

				eStatus	:= Done;

			END_IF

		MagConv2ClpActRmtClprSetUnclamp:
			IF eStatus = Idle OR eStatus = Busy THEN

				eStatus	:= Busy;

				bMtrSigOnOrLToR	:= FALSE;
				bMtrDirOrRToL	:= FALSE;

				bRmtClprClampCtrl	:= FALSE;

				eStatus	:= Done;

			END_IF

		MagConv2ClpActRmtClprClamp:
			IF eStatus = Idle OR eStatus = Busy THEN

				eStatus	:= Busy;

				bMtrSigOnOrLToR	:= FALSE;
				bMtrDirOrRToL	:= FALSE;

				bRmtClprClampCtrl	:= TRUE;

				fbRmtClprClampChk.bExtSen		:= p_bRmtClprClampSen;
				fbRmtClprClampChk.bRetSen		:= p_bRmtClprUnclampSen;
				fbRmtClprClampChk.bExtSafety	:= p_bRmtClprClampSafetySen;
				fbRmtClprClampChk(bEn := TRUE);

				IF fbRmtClprClampChk.udiStatus = 0 THEN
					eStatus	:= Done;
				ELSIF fbRmtClprClampChk.udiStatus < 65534 THEN
					bRmtClprClampCtrl	:= FALSE;

					eStatus	:= Error;

					IF fbRmtClprClampChk.udiStatus = 1503 THEN
						udiStatus	:= 10016;	//Clamper Clamp Sensor On Time Out In Clamp Check While Clamper Clamp
					ELSIF fbRmtClprClampChk.udiStatus = 1506 THEN
						udiStatus	:= 10017;	//Clamper Unclamp Sensor Off Time Out In Clamp Check While Clamper Clamp
					ELSIF fbRmtClprClampChk.udiStatus = 1507 THEN
						udiStatus	:= 10018;	//Clamper Clamp Safety Sensor Error In Clamp Check While Clamper Clamp
					ELSE
						udiStatus	:= fbRmtClprClampChk.udiStatus;
					END_IF
				END_IF
			END_IF

		MagConv2ClpActRmtClprUnclamp:
			IF eStatus = Idle OR eStatus = Busy THEN

				eStatus	:= Busy;

				bMtrSigOnOrLToR	:= FALSE;
				bMtrDirOrRToL	:= FALSE;

				bRmtClprClampCtrl	:= FALSE;

				fbRmtClprUnclampChk.bExtSen		:= p_bRmtClprClampSen;
				fbRmtClprUnclampChk.bRetSen		:= p_bRmtClprUnclampSen;
				fbRmtClprUnclampChk.bRetSafety	:= p_bRmtClprUnclampSafetySen;
				fbRmtClprUnclampChk(bEn := TRUE);

				IF fbRmtClprUnclampChk.udiStatus = 0 THEN
					eStatus	:= Done;
				ELSIF fbRmtClprUnclampChk.udiStatus < 65534 THEN
					bRmtClprClampCtrl	:= TRUE;

					eStatus	:= Error;

					IF fbRmtClprUnclampChk.udiStatus = 1504 THEN
						udiStatus	:= 10019;	//Clamper Clamp Sensor Off Time Out In Unclamp Check While Clamper Unclamp
					ELSIF fbRmtClprUnclampChk.udiStatus = 1505 THEN
						udiStatus	:= 10020;	//Clamper Unclamp Sensor On Time Out In Unclamp Check While Clamper Unclamp
					ELSIF fbRmtClprUnclampChk.udiStatus = 1508 THEN
						udiStatus	:= 10021;	//Clamper Unclamp Safety Sensor Error In Unclamp Check While Clamper Unclamp
					ELSE
						udiStatus	:= fbRmtClprUnclampChk.udiStatus;
					END_IF
				END_IF

			END_IF

		MagConv2ClpActStop:
			IF eStatus = Idle OR eStatus = Busy THEN

				eStatus	:= Busy;

				//Conveyor Run
				fbStop(bEn := TRUE);

				bMtrSigOnOrLToR	:= fbStop.bMtrSigOnOrLToR;
				bMtrDirOrRToL	:= fbStop.bMtrDirOrRToL;

				IF fbStop.udiStatus = 0 THEN
					eStatus	:= Done;
				ELSIF fbStop.udiStatus < 65534 THEN
					udiStatus	:= fbStop.udiStatus;
					eStatus		:= Error;
				END_IF

			END_IF

		MagConv2ClpActStopClpr:
			IF eStatus = Idle OR eStatus = Busy THEN

				eStatus	:= Busy;

				//Conveyor Run
				fbStop(bEn := TRUE);

				bMtrSigOnOrLToR	:= fbStop.bMtrSigOnOrLToR;
				bMtrDirOrRToL	:= fbStop.bMtrDirOrRToL;

				bFixClprClampCtrl	:= FALSE;
				bRmtClprClampCtrl	:= FALSE;

				fbFixClprUnclampChk.bExtSen		:= p_bFixClprClampSen;
				fbFixClprUnclampChk.bRetSen		:= p_bFixClprUnclampSen;
				fbFixClprUnclampChk.bRetSafety	:= p_bFixClprUnclampSafetySen;
				fbFixClprUnclampChk(bEn := TRUE);

				fbRmtClprUnclampChk.bExtSen		:= p_bRmtClprClampSen;
				fbRmtClprUnclampChk.bRetSen		:= p_bRmtClprUnclampSen;
				fbRmtClprUnclampChk.bRetSafety	:= p_bRmtClprUnclampSafetySen;
				fbRmtClprUnclampChk(bEn := TRUE);

				IF fbStop.udiStatus = 0 AND fbFixClprUnclampChk.udiStatus = 0 AND fbRmtClprUnclampChk.udiStatus = 0 THEN
					eStatus		:= Done;
				ELSIF fbStop.udiStatus > 0 AND fbStop.udiStatus < 65534 THEN
					udiStatus	:= fbStop.udiStatus;
					eStatus		:= Error;
				ELSIF (fbFixClprUnclampChk.udiStatus > 0 AND fbFixClprUnclampChk.udiStatus < 65534) OR (fbRmtClprUnclampChk.udiStatus > 0 AND fbRmtClprUnclampChk.udiStatus < 65534) THEN
					bFixClprClampCtrl	:= TRUE;
					bRmtClprClampCtrl	:= TRUE;

					eStatus	:= Error;

					IF fbFixClprUnclampChk.udiStatus = 1504 OR fbRmtClprUnclampChk.udiStatus = 1504 THEN
						udiStatus	:= 10022;	//Clamper Clamp Sensor Off Time Out In Unclamp Check While Stop With Clamper
					ELSIF fbFixClprUnclampChk.udiStatus = 1505 OR fbRmtClprUnclampChk.udiStatus = 1505 THEN
						udiStatus	:= 10023;	//Clamper Unclamp Sensor On Time Out In Unclamp Check While Stop With Clamper
					ELSIF fbFixClprUnclampChk.udiStatus = 1508 OR fbRmtClprUnclampChk.udiStatus = 1508 THEN
						udiStatus	:= 10024;	//Clamper Unclamp Safety Sensor Error In Unclamp Check While Stop With Clamper
					ELSE
						IF fbFixClprUnclampChk.udiStatus > 0 AND fbFixClprUnclampChk.udiStatus < 65534 THEN
							udiStatus	:= fbFixClprUnclampChk.udiStatus;
						ELSIF fbRmtClprUnclampChk.udiStatus > 0 AND fbRmtClprUnclampChk.udiStatus < 65534 THEN
							udiStatus	:= fbRmtClprUnclampChk.udiStatus;
						END_IF
					END_IF
				END_IF

			END_IF

		MagConv2ClpActSetMtrSigOnOrLToR:
			IF eStatus = Idle OR eStatus = Busy THEN

				bMtrSigOnOrLToR	:= TRUE;

				eStatus	:= Done;

			END_IF

		MagConv2ClpActSetMtrDirOrRToL:
			IF eStatus = Idle OR eStatus = Busy THEN

				bMtrDirOrRToL	:= TRUE;

				eStatus	:= Done;

			END_IF

		MagConv2ClpActRstMtrSigOnOrLToR:
			IF eStatus = Idle OR eStatus = Busy THEN

				bMtrSigOnOrLToR	:= FALSE;

				eStatus	:= Done;

			END_IF

		MagConv2ClpActRstMtrDirOrRToL:
			IF eStatus = Idle OR eStatus = Busy THEN

				bMtrDirOrRToL	:= FALSE;

				eStatus	:= Done;

			END_IF

		MagConv2ClpActSetMtrAll:
			IF eStatus = Idle OR eStatus = Busy THEN

				bMtrSigOnOrLToR	:= TRUE;
				bMtrDirOrRToL	:= TRUE;

				eStatus	:= Done;

			END_IF

		MagConv2ClpActRstMtrAll:
			IF eStatus = Idle OR eStatus = Busy THEN

				bMtrSigOnOrLToR	:= FALSE;
				bMtrDirOrRToL	:= FALSE;

				eStatus	:= Done;

			END_IF

	END_CASE

END_ACTION
```

#### InputRef.var - Do Not Change!!!
```iecst
(*2019-10-30*)
(**)
(*General*)
VAR
	p_eAct : REFERENCE TO eMagConv2ClpAction;
	p_udiRstErr : REFERENCE TO UDINT;
	p_bPrep : REFERENCE TO BOOL;
	p_bEn : REFERENCE TO BOOL;
	p_bDis : REFERENCE TO BOOL;
END_VAR
(**)
(*Configuration*)
VAR
	p_bManual : REFERENCE TO BOOL;
	p_bOnDirMod : REFERENCE TO BOOL;
	p_diInitTm : REFERENCE TO DINT;
	p_tMtrOffDlyTm : REFERENCE TO TIME;
	p_diTxInTimeOut : REFERENCE TO DINT;
	p_diTxOutTimeOut : REFERENCE TO DINT;
	p_eDirection : REFERENCE TO eConvDir;
	p_sProgNm : REFERENCE TO STRING[15];
	p_tClprClampTO : REFERENCE TO TIME;
	p_tClprUnclampTO : REFERENCE TO TIME;
	p_bNtSettingsLoadDone : REFERENCE TO BOOL;
END_VAR
(**)
(*Input*)
VAR
	p_bLeftSen : REFERENCE TO BOOL;
	p_bRightSen : REFERENCE TO BOOL;
	p_bFixClprClampSen : REFERENCE TO BOOL;
	p_bFixClprUnclampSen : REFERENCE TO BOOL;
	p_bRmtClprClampSen : REFERENCE TO BOOL;
	p_bRmtClprUnclampSen : REFERENCE TO BOOL;
	p_bFixClprClampSafetySen : REFERENCE TO BOOL;
	p_bFixClprUnclampSafetySen : REFERENCE TO BOOL;
	p_bRmtClprClampSafetySen : REFERENCE TO BOOL;
	p_bRmtClprUnclampSafetySen : REFERENCE TO BOOL;
	p_bWidthChkSen : REFERENCE TO BOOL;
	p_bWidthChkSenPrep : REFERENCE TO BOOL;
	p_bWidthChkInterrupt : REFERENCE TO BOOL;
END_VAR
```

#### Local.var - Do Not Change!!!
```iecst
(*2019-10-30*)
VAR
	tylocalMagConv2Clp : tyMagConv2Clp;
END_VAR
(**)
(*Local Action, State & Status*)
VAR
	eAct : eMagConv2ClpAction := MagConv2ClpActIdle;
	udiStatus : UDINT := 0;
	a_sStatText : ARRAY[0..50] OF STRING[200] := ['Idling','Initializing','Initializing With Stop Then Clamper','Initializing With Clamper Then Stop','Entering Board','Entering Board With Stop Then Clamper','Entering Board With Clamper Then Stop','Pre-Exiting Board','Pre-Exiting Board With Clamper',2('Exiting Board'),2('Exiting Board With Clamper'),'Fix/Bottom Clamper Setting All Control','Fix/Bottom Clamper Resetting All Control','Fix/Bottom Clamper Setting Clamp','Fix/Bottom Clamper Setting Unclamp','Fix/Bottom Clamper Clamp','Fix/Bottom Clampler Unclamp','Remote/Top Clamper Setting All Control','Remote/Top Clamper Resetting All Control','Remote/Top Clamper Setting Clamp','Remote/Top Clamper Setting Unclamp','Remote/Top Clamper Clamp','Remote/Top Clampler Unclamp','Stopping','Stopping With Clamper','Turning On Motor Signal','Turning On Motor Direction','Turning Off Motor Signal','Turning Off Motor Direction','Turning On All Motor Output','Turning Off All Motor Output',18('')];
END_VAR
(**)
(*Local Alarm*)
VAR
	tyAlmData : tyAlmDat;
END_VAR
(**)
(*Local Output*)
VAR
	bHvMag : BOOL := FALSE;
	bMtrSigOnOrLToR : BOOL := FALSE;
	bMtrDirOrRToL : BOOL := FALSE;
	bFixClprClampCtrl : BOOL;
	bRmtClprClampCtrl : BOOL;
	bClprTwoOutputControl : BOOL := FALSE;
END_VAR
(**)
(*Local Input*)
VAR
	udiRstErr : UDINT := 0;
	bPrep : BOOL := TRUE;
	bEn : BOOL := TRUE;
	bDis : BOOL := FALSE;
	bManual : BOOL := FALSE;
	bOnDirMod : BOOL := FALSE;
	diInitTm : DINT := 10000;
	tMtrOffDlyTm : TIME := T#0S;
	diTxInTimeOut : DINT := 10000;
	diTxOutTimeOut : DINT := 10000;
	eDirection : eConvDir := ConvDirLToR;
	bLeftSen : BOOL := FALSE;
	bRightSen : BOOL := FALSE;
	bFixClprClampSen : BOOL := FALSE;
	bFixClprUnclampSen : BOOL := FALSE;
	bFixClprClampSafetySen : BOOL := TRUE;
	bFixClprUnclampSafetySen : BOOL := TRUE;
	bRmtClprClampSen : BOOL := FALSE;
	bRmtClprUnclampSen : BOOL := FALSE;
	bRmtClprClampSafetySen : BOOL := TRUE;
	bRmtClprUnclampSafetySen : BOOL := TRUE;
	bWidthChkPrep : BOOL := TRUE;
	sProgNm : STRING[15] := 'MagConv2Clp';
	tClprClampTO : TIME := T#20s;
	tClprUnclampTO : TIME := T#20s;
	bNtSettingsLoadDone : BOOL := TRUE;
END_VAR
(**)
(*Local*)
VAR
	bRstErr : BOOL;
	udiRstErrOld : UDINT;
	bInitDone : BOOL;
	bInitialDone : BOOL;
	bReachEnd : BOOL;
	usiStep : USINT;
	usiSubStep : USINT;
	eStatOld : eMagConv2ClpAction := MagConv2ClpActIdle;
	fbInit : fbConvSenToSenTm;
	fbEnt : fbConvSenToSen;
	fbPreExit : fbConvSenToSenTm;
	fbExit : fbConvSenToSenOff;
	fbExit1 : fbConvSenToSenOff1;
	fbStop : fbConvMtrOff;
	fbFixClprClampChk : fbPneuExtRetSenExtChk;
	fbFixClprUnclampChk : fbPneuExtRetSenRetChk;
	fbRmtClprClampChk : fbPneuExtRetSenExtChk;
	fbFixClprDly : TON := (PT:=T#1s);
	fbRmtClprUnclampChk : fbPneuExtRetSenRetChk;
	fbClprDlyTm : TON;
	fbSmallLargeSenDlyTm : TON := (PT:=T#1S);
	fbWidthChk : TON := (PT:=T#30s);
	fbLeftSenDelayTm : TON := (PT:=T#1S);
	fbFixClpExtChkTm : TON := (PT:=T#5s);
	fbRmtClpExtChkTm : TON := (PT:=T#3s);
	udiModuleNum : UDINT := 1901;
END_VAR
(**)
VAR
	bMag1FixedClampCtrl : BOOL;
	bMag2FixedClampCtrl : BOOL;
	bMag1ConvMtrIn : BOOL;
	bMag1ConvMtrOut : BOOL;
	bMag2ConvMtrIn : BOOL;
	bMag2ConvMtrOut : BOOL;
END_VAR
```

#### Act_InputConfig.st - not listed in the package file held
```iecst
(** 2019-10-30 **)
ACTION Act_InputConfig:

	(* Always Change If Project Change *)

	//Pass Data To Link

	tylocalMagConv2Clp.In.bLinkDISafetyRlySig := g_tyDInput.bSafetyRlySig;

	tylocalMagConv2Clp.In.bLinkMagSmallSen := g_tyDInput.bMagConvSmallMagSen1;
	tylocalMagConv2Clp.In.bLinkMagLargeSen := g_tyDInput.bMagConvLargeMagSen1;
	tylocalMagConv2Clp.In.bLinkFixClprUnClampSen := g_tyDInput.bMag1FixedUnclampRS;
//	tylocalMagConv2Clp.In.bLinkFixClprClampSen := g_tyDInput.bMag1FixedClampRS; // Pneumatic Clamp Reed Switch
	tylocalMagConv2Clp.In.bLinkFixClprMagDetectSen := g_tyDInput.bMag1FixedClampSen; // Clamping Done Before Pneumatic Clamp Reed Switch for special Condition
	tylocalMagConv2Clp.In.bLinkFixClprMagDetectSenPrep := g_tyNtParamCurr.bProjFixClpMagDSenPrep; // Fixed Clamp Detect Sensor Prep before Clamp RS

	tylocalMagConv2Clp.In.bLinkMagOpsStepMagFullExit := g_tyOpsMagConvUL1MagFullExit;
	tylocalMagConv2Clp.In.bLinkDIMagEntSen := g_tyDInput.bMagConvEntSen1;
//	tylocalMagConv2Clp.In.bLinkDO := g_tyDO;

	tylocalMagConv2Clp.In.bWidthChkSen := g_tyNtParamCurr.bCurtainSenPrep;
	tylocalMagConv2Clp.In.bWidthChkInterrupt := g_tyDInput.bCurtainSen;

	tylocalMagConv2Clp.In.bLinkNtParamMagModelAutoVerify := g_tyNtParamCurr.bProjMagAutoVerifyPrep;
//	tylocalMagConv2Clp.In.tyDISettings := g_tyNtParamCurr.tyDISettings;
//	tylocalMagConv2Clp.In.bLinkFixClprClampSen ACCESS ADR(bFixClprClampSen);//tylocalMagConv2Clp.In.DIMag1FixedSideDetect;//tylocalMagConv2Clp.In.DIMag1FixedClampRS; //initLocal at 1st

	//Pass Data To Internal Use
	tylocalMagConv2Clp.In.udiRstErr := g_tyRstErrReset;
	tylocalMagConv2Clp.In.bPrep := g_tyNtParamCurr.bProjMag1ConvPrep;
	tylocalMagConv2Clp.In.bManual := g_tyUIMnlMod;
	tylocalMagConv2Clp.In.bOnDirMod := g_tyNtParamCurr.bMagConv1OnDirMod;
	tylocalMagConv2Clp.In.diInitTm := g_tyMcParamCurr.tMag1ConvRunTmOut;
	tylocalMagConv2Clp.In.tMtrOffDlyTm := g_tyNtParamCurr.tMagConv1MtrOffDlyTm;
	tylocalMagConv2Clp.In.diTxInTimeOut := g_tyMcParamCurr.tMag1ConvRunTmOut;
	tylocalMagConv2Clp.In.diTxOutTimeOut := g_tyMcParamCurr.tMag1ConvRunTmOut;
	tylocalMagConv2Clp.In.eDirection := g_tyNtParamCurr.bProjMagConvDir;
	tylocalMagConv2Clp.In.sProgNm := g_tyNtParamCurr.sMagConv1ProgNm;
	tylocalMagConv2Clp.In.tClprClampTO := g_tyNtParamCurr.tMagConv1ClprClampTO;
	tylocalMagConv2Clp.In.tClprUnclampTO := g_tyNtParamCurr.tMagConv1ClprUnclampTO;
//	tylocalMagConv2Clp.In.bLeftSen := g_tyDInput.bMagPresentSen1;
	tylocalMagConv2Clp.In.bRightSen	:= g_tyDInput.bMagPresentSen1;

	(* Always Change If Project Change *)

	IF g_tyOps.bRun THEN
		tylocalMagConv2Clp.In.eAct := g_tyOpsMagConvUL1.eMagConv2ClpAct;
	ELSIF tylocalMagConv2Clp.In.bManual = TRUE THEN
		tylocalMagConv2Clp.In.eAct := g_tyUIOut.eMnlAct.eMagConv2Clp1Act;
	ELSE
		tylocalMagConv2Clp.In.eAct := eAct;
	END_IF
END_ACTION
```

#### Act_OutputConfig.st - not listed in the package file held
```iecst
ACTION Act_OutputConfig:
	// Output: Assign To Global For Independent Package Usage

	g_tyPneuMag3AWEngage := tylocalMagConv2Clp.Out; // Change the Global Naming According to the Physical Hardware Module

END_ACTION
```

### Program Logical/MagConv_LiftnTrav/MagConv2Clp2 (IEC) - 1.00.0 - NtConv v5.00.0 , NtPneu v5.00.0

#### InputRef_Link.var
```iecst
(*2019-10-30*)
(**)
VAR
	p_bLinkOpsRun : REFERENCE TO BOOL;
END_VAR
(**)
VAR
	p_bLinkDISafetyRlySig : REFERENCE TO BOOL;
	p_bLinkMagSmallSen : REFERENCE TO BOOL;
	p_bLinkMagLargeSen : REFERENCE TO BOOL;
	p_bLinkFixClprUnClampSen : REFERENCE TO BOOL;
	p_bLinkFixClprClampSen : REFERENCE TO BOOL;
	p_bLinkFixClprMagDetectSen : REFERENCE TO BOOL;
	p_bLinkFixClprMagDetectSenPrep : REFERENCE TO BOOL;
	p_bLinkMagOpsStepMagFullExit : REFERENCE TO BOOL;
	p_bLinkDIMagEntSen : REFERENCE TO BOOL;
	p_bLinkDO : REFERENCE TO tyDigitalOutput;
	p_bLinkNtParamMagModelAutoVerify : REFERENCE TO BOOL;
	p_tyDISettings : REFERENCE TO tyDigitalInputSettings;
END_VAR
```
